KUKA KRL program: MyProgram_209().src

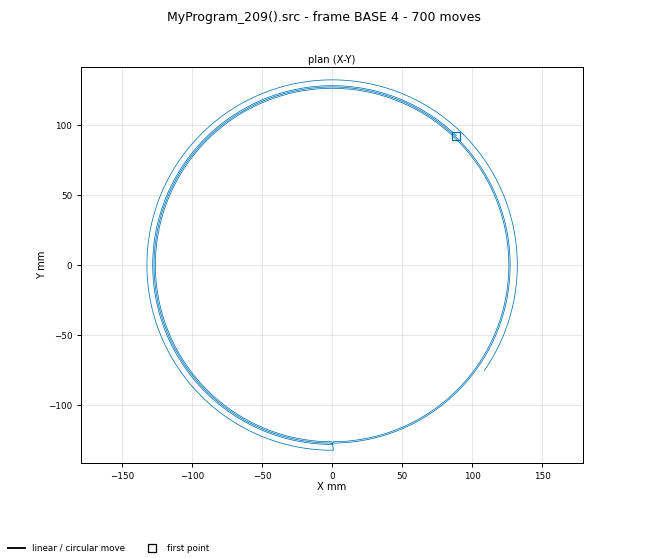
[picture p0: tool path of MyProgram_209().src in frame BASE 4, 700 of 700 moves have a stored position in this frame; points joined in program order, loops and branches not executed]
&ACCESS RVP
&REL 1
&PARAM TEMPLATE = C:\KRC\Roboter\Template\vorgabe
&PARAM EDITMASK = *
DEF MyProgram_209()
; ---- Setting reference (Base) ----
$BASE = BASE_DATA[4]

; --------------------------
; ---- Setting tool (TCP) ----
$TOOL = TOOL_DATA[3]
; --------------------------

$VEL.CP = VEL_APROX_PRINT
Startdeposition()
$VEL.CP = VEL_PRINT
LIN {X 88.7126,Y 92.477,Z 148,A 43.8343,B 21.8486,C -1.1424,E1 21.9863,E2 403.3687} C_DIS
LIN {X 86.374,Y 94.6653,Z 148,A 45.08,B 21.8488,C -1.1368,E1 21.9838,E2 402.1439} C_DIS
LIN {X 83.0937,Y 97.5567,Z 148,A 47.0034,B 21.8488,C -1.1392,E1 21.9797,E2 400.2228} C_DIS
LIN {X 79.622,Y 100.4104,Z 148,A 48.9944,B 21.8486,C -1.1421,E1 21.9754,E2 398.2327} C_DIS
LIN {X 76.1775,Y 103.0485,Z 148,A 50.9778,B 21.8483,C -1.1475,E1 21.971,E2 396.243} C_DIS
LIN {X 72.5158,Y 105.6566,Z 148,A 52.8915,B 21.8483,C -1.1466,E1 21.9666,E2 394.3396} C_DIS
LIN {X 68.9845,Y 107.9954,Z 148,A 54.8188,B 21.8481,C -1.1511,E1 21.9621,E2 392.4074} C_DIS
LIN {X 64.9135,Y 110.4902,Z 148,A 56.7473,B 21.8484,C -1.1451,E1 21.9575,E2 390.5022} C_DIS
LIN {X 61.7494,Y 112.2898,Z 148,A 58.5868,B 21.8478,C -1.1569,E1 21.953,E2 388.6373} C_DIS
LIN {X 58.4226,Y 114.0537,Z 148,A 60.0443,B 21.8482,C -1.149,E1 21.9494,E2 387.2056} C_DIS
LIN {X 55.5123,Y 115.4982,Z 148,A 61.5938,B 21.8479,C -1.1551,E1 21.9455,E2 385.6445} C_DIS
LIN {X 52.3493,Y 116.9655,Z 148,A 63.1517,B 21.8479,C -1.1569,E1 21.9416,E2 384.0863} C_DIS
LIN {X 47.2118,Y 119.1343,Z 148,A 65.6144,B 21.8478,C -1.1582,E1 21.9352,E2 381.627} C_DIS
LIN {X 43.1467,Y 120.6643,Z 148,A 67.6588,B 21.8474,C -1.1646,E1 21.9298,E2 379.5704} C_DIS
LIN {X 39.1405,Y 122.0223,Z 148,A 69.483,B 21.8475,C -1.1632,E1 21.925,E2 377.7539} C_DIS
LIN {X 35.9508,Y 122.9998,Z 148,A 70.9408,B 21.8475,C -1.1628,E1 21.9211,E2 376.3001} C_DIS
LIN {X 32.7097,Y 123.9016,Z 148,A 72.5384,B 21.8473,C -1.168,E1 21.9168,E2 374.6917} C_DIS
LIN {X 28.571,Y 124.9205,Z 148,A 74.3,B 21.8475,C -1.1627,E1 21.9121,E2 372.947} C_DIS
LIN {X 25.5331,Y 125.5767,Z 148,A 75.7516,B 21.8474,C -1.1661,E1 21.9081,E2 371.4884} C_DIS
LIN {X 21.7512,Y 126.2885,Z 148,A 77.403,B 21.8474,C -1.1638,E1 21.9036,E2 369.8455} C_DIS
LIN {X 17.695,Y 126.9194,Z 148,A 79.2772,B 21.8474,C -1.1661,E1 21.8984,E2 367.9672} C_DIS
LIN {X 12.2711,Y 127.5574,Z 148,A 81.7514,B 21.8473,C -1.1679,E1 21.8915,E2 365.49} C_DIS
LIN {X 8.4289,Y 127.87,Z 148,A 83.6291,B 21.8469,C -1.1747,E1 21.8862,E2 363.5952} C_DIS
LIN {X 3.9153,Y 128.0871,Z 148,A 86.0268,B 21.8461,C -1.191,E1 21.8794,E2 361.1544} C_DIS
LIN {X -0.4369,Y 128.146,Z 148,A 87.4571,B 21.8473,C -1.1683,E1 21.8756,E2 359.785} C_DIS
LIN {X -3.2199,Y 128.1064,Z 148,A 89.2919,B 21.846,C -1.1935,E1 21.8703,E2 357.8824} C_DIS
LIN {X -7.9141,Y 127.9018,Z 148,A 90.7155,B 21.8475,C -1.1636,E1 21.8665,E2 356.5386} C_DIS
LIN {X -13.7506,Y 127.4064,Z 148,A 93.443,B 21.8473,C -1.167,E1 21.8589,E2 353.8004} C_DIS
LIN {X -17.7931,Y 126.9054,Z 148,A 95.2356,B 21.8474,C -1.1647,E1 21.854,E2 352.0124} C_DIS
LIN {X -21.7145,Y 126.2946,Z 148,A 97.2457,B 21.847,C -1.1735,E1 21.8483,E2 349.9764} C_DIS
LIN {X -26.441,Y 125.3901,Z 148,A 99.2681,B 21.8474,C -1.1663,E1 21.8429,E2 347.9708} C_DIS
LIN {X -30.0308,Y 124.5776,Z 148,A 100.8142,B 21.8476,C -1.1607,E1 21.8387,E2 346.4374} C_DIS
LIN {X -33.5956,Y 123.6653,Z 148,A 102.571,B 21.8475,C -1.1638,E1 21.8339,E2 344.6693} C_DIS
LIN {X -37.953,Y 122.3977,Z 148,A 105.1421,B 21.8464,C -1.1845,E1 21.8269,E2 342.0373} C_DIS
LIN {X -42.6562,Y 120.8402,Z 148,A 106.8737,B 21.8476,C -1.1614,E1 21.8225,E2 340.364} C_DIS
LIN {X -46.3756,Y 119.46,Z 148,A 108.4825,B 21.8481,C -1.1522,E1 21.8183,E2 338.776} C_DIS
LIN {X -49.6081,Y 118.1544,Z 148,A 110.1026,B 21.8481,C -1.1526,E1 21.8141,E2 337.1506} C_DIS
LIN {X -52.9938,Y 116.6772,Z 148,A 111.8643,B 21.8479,C -1.1548,E1 21.8096,E2 335.3781} C_DIS
LIN {X -56.5469,Y 114.9949,Z 148,A 113.4646,B 21.8484,C -1.1456,E1 21.8056,E2 333.7978} C_DIS
LIN {X -58.9703,Y 113.7731,Z 148,A 114.9346,B 21.848,C -1.1543,E1 21.8019,E2 332.2999} C_DIS
LIN {X -65.619,Y 110.0727,Z 148,A 117.9071,B 21.8491,C -1.1306,E1 21.7949,E2 329.381} C_DIS
LIN {X -68.3515,Y 108.3971,Z 148,A 119.6031,B 21.8487,C -1.1388,E1 21.7907,E2 327.6567} C_DIS
LIN {X -71.7262,Y 106.1943,Z 148,A 121.3334,B 21.8491,C -1.1324,E1 21.7867,E2 325.937} C_DIS
LIN {X -74.857,Y 104.0117,Z 148,A 123.0427,B 21.8492,C -1.1292,E1 21.7828,E2 324.2296} C_DIS
LIN {X -78.0018,Y 101.6738,Z 148,A 125.0863,B 21.8488,C -1.1375,E1 21.7782,E2 322.1549} C_DIS
LIN {X -82.0467,Y 98.4396,Z 148,A 127.2208,B 21.8494,C -1.1251,E1 21.7737,E2 320.0446} C_DIS
LIN {X -84.4392,Y 96.3947,Z 148,A 128.6876,B 21.8494,C -1.1245,E1 21.7706,E2 318.5729} C_DIS
LIN {X -86.7423,Y 94.3273,Z 148,A 130.143,B 21.8494,C -1.1242,E1 21.7675,E2 317.1113} C_DIS
LIN {X -90.1509,Y 91.0754,Z 148,A 132.2112,B 21.8498,C -1.1177,E1 21.7634,E2 315.0505} C_DIS
LIN {X -93.4013,Y 87.739,Z 148,A 134.2865,B 21.85,C -1.1124,E1 21.7594,E2 312.9793} C_DIS
LIN {X -96.9151,Y 83.8411,Z 148,A 136.6811,B 21.8502,C -1.1085,E1 21.755,E2 310.5828} C_DIS
LIN {X -99.8508,Y 80.3225,Z 148,A 139.056,B 21.8498,C -1.1165,E1 21.7507,E2 308.1735} C_DIS
LIN {X -102.2342,Y 77.266,Z 148,A 140.2541,B 21.8511,C -1.0902,E1 21.7488,E2 307.0397} C_DIS
LIN {X -105.1847,Y 73.1985,Z 148,A 142.6997,B 21.8511,C -1.0921,E1 21.7448,E2 304.5749} C_DIS
LIN {X -107.6475,Y 69.5268,Z 148,A 144.6782,B 21.8513,C -1.0867,E1 21.7418,E2 302.5995} C_DIS
LIN {X -111.8681,Y 62.51,Z 148,A 148.3886,B 21.8517,C -1.0783,E1 21.7365,E2 298.8896} C_DIS
LIN {X -113.501,Y 59.4885,Z 148,A 150.8638,B 21.8501,C -1.112,E1 21.7332,E2 296.3079} C_DIS
LIN {X -116.4877,Y 53.4055,Z 148,A 153.0192,B 21.8522,C -1.0675,E1 21.7308,E2 294.2592} C_DIS
LIN {X -118.1611,Y 49.5922,Z 148,A 154.7522,B 21.8527,C -1.0567,E1 21.7289,E2 292.5442} C_DIS
LIN {X -119.4347,Y 46.4407,Z 148,A 157.2556,B 21.851,C -1.0919,E1 21.7263,E2 289.9294} C_DIS
LIN {X -121.6112,Y 40.3995,Z 148,A 160.267,B 21.8512,C -1.0887,E1 21.7236,E2 286.9066} C_DIS
LIN {X -123.6546,Y 33.6359,Z 148,A 162.4583,B 21.8534,C -1.0396,E1 21.722,E2 284.8333} C_DIS
LIN {X -124.5826,Y 30.01,Z 148,A 164.021,B 21.8539,C -1.03,E1 21.721,E2 283.286} C_DIS
LIN {X -125.2863,Y 26.9219,Z 148,A 165.5058,B 21.8539,C -1.0283,E1 21.7201,E2 281.7957} C_DIS
LIN {X -126.0639,Y 23.0116,Z 148,A 167.3491,B 21.8541,C -1.025,E1 21.7191,E2 279.9485} C_DIS
LIN {X -126.7094,Y 19.1419,Z 148,A 169.1664,B 21.8542,C -1.022,E1 21.7183,E2 278.1269} C_DIS
LIN {X -127.217,Y 15.4067,Z 148,A 170.7737,B 21.8546,C -1.0135,E1 21.7178,E2 276.5314} C_DIS
LIN {X -127.626,Y 11.5569,Z 148,A 172.6352,B 21.8546,C -1.0132,E1 21.7173,E2 274.6577} C_DIS
LIN {X -127.9165,Y 7.6748,Z 148,A 174.3037,B 21.855,C -1.0047,E1 21.717,E2 273.0003} C_DIS
LIN {X -128.0928,Y 3.7093,Z 148,A 176.0592,B 21.8553,C -0.9983,E1 21.7168,E2 271.2501} C_DIS
LIN {X -128.1496,Y -0.0528,Z 148,A 178.0622,B 21.8549,C -1.0058,E1 21.7168,E2 269.2128} C_DIS
LIN {X -128.0484,Y -5.0106,Z 148,A -179.9662,B 21.8557,C -0.9889,E1 21.7169,E2 267.2731} C_DIS
LIN {X -127.8019,Y -9.389,Z 148,A -178.0277,B 21.856,C -0.9818,E1 21.7173,E2 265.3402} C_DIS
LIN {X -127.4676,Y -13.1819,Z 148,A -176.2505,B 21.856,C -0.9794,E1 21.7177,E2 263.5571} C_DIS
LIN {X -127.0317,Y -16.8659,Z 148,A -174.6426,B 21.8564,C -0.9721,E1 21.7183,E2 261.9576} C_DIS
LIN {X -126.4164,Y -20.9847,Z 148,A -172.7768,B 21.8566,C -0.9665,E1 21.7191,E2 260.0942} C_DIS
LIN {X -125.7225,Y -24.8164,Z 148,A -170.9204,B 21.8566,C -0.9657,E1 21.7201,E2 258.2272} C_DIS
LIN {X -124.9393,Y -28.4888,Z 148,A -169.3254,B 21.857,C -0.9572,E1 21.721,E2 256.6442} C_DIS
LIN {X -124.0092,Y -32.3059,Z 148,A -167.6182,B 21.8573,C -0.9498,E1 21.7222,E2 254.9454} C_DIS
LIN {X -123.3197,Y -34.8394,Z 148,A -166.2083,B 21.8571,C -0.9558,E1 21.7233,E2 253.5098} C_DIS
LIN {X -122.1023,Y -38.8901,Z 148,A -164.4411,B 21.8575,C -0.9451,E1 21.7247,E2 251.7596} C_DIS
LIN {X -120.0335,Y -44.8704,Z 148,A -161.7574,B 21.8581,C -0.9309,E1 21.7272,E2 249.0967} C_DIS
LIN {X -118.8089,Y -48.0192,Z 148,A -160.1373,B 21.8581,C -0.9309,E1 21.7289,E2 247.4659} C_DIS
LIN {X -117.5359,Y -51.0561,Z 148,A -158.593,B 21.8581,C -0.9297,E1 21.7306,E2 245.9152} C_DIS
LIN {X -115.7831,Y -54.9159,Z 148,A -156.6975,B 21.8584,C -0.9243,E1 21.7328,E2 244.0221} C_DIS
LIN {X -114.2963,Y -57.9462,Z 148,A -155.3639,B 21.8588,C -0.913,E1 21.7344,E2 242.7107} C_DIS
LIN {X -112.3675,Y -61.6074,Z 148,A -153.2902,B 21.8587,C -0.917,E1 21.7372,E2 240.6134} C_DIS
LIN {X -110.1286,Y -65.5253,Z 148,A -151.2391,B 21.8588,C -0.913,E1 21.7401,E2 238.5607} C_DIS
LIN {X -107.9003,Y -69.1332,Z 148,A -149.3445,B 21.859,C -0.908,E1 21.7429,E2 236.6684} C_DIS
LIN {X -105.4709,Y -72.7864,Z 148,A -147.3415,B 21.8591,C -0.9048,E1 21.746,E2 234.6627} C_DIS
LIN {X -103.0791,Y -76.1358,Z 148,A -145.2043,B 21.8588,C -0.9125,E1 21.7496,E2 232.4926} C_DIS
LIN {X -100.9621,Y -78.9203,Z 148,A -143.8505,B 21.8593,C -0.9001,E1 21.7519,E2 231.165} C_DIS
LIN {X -97.9265,Y -82.6583,Z 148,A -141.7279,B 21.8596,C -0.8938,E1 21.7557,E2 229.0479} C_DIS
LIN {X -94.8508,Y -86.1696,Z 148,A -139.6882,B 21.8598,C -0.8871,E1 21.7594,E2 227.0156} C_DIS
LIN {X -91.854,Y -89.3577,Z 148,A -137.6716,B 21.8599,C -0.8854,E1 21.7633,E2 224.9936} C_DIS
LIN {X -88.8005,Y -92.3929,Z 148,A -135.7075,B 21.8599,C -0.883,E1 21.7673,E2 223.0264} C_DIS
LIN {X -85.5251,Y -95.4322,Z 148,A -133.7701,B 21.8602,C -0.8765,E1 21.7712,E2 221.0975} C_DIS
LIN {X -82.2328,Y -98.2836,Z 148,A -131.8219,B 21.8604,C -0.8728,E1 21.7754,E2 219.1505} C_DIS
LIN {X -78.9585,Y -100.9331,Z 148,A -129.8981,B 21.8604,C -0.871,E1 21.7796,E2 217.2231} C_DIS
LIN {X -76.531,Y -102.7855,Z 148,A -128.228,B 21.8601,C -0.8814,E1 21.7834,E2 215.5179} C_DIS
LIN {X -73.5721,Y -104.9244,Z 148,A -126.8123,B 21.8605,C -0.8696,E1 21.7866,E2 214.1286} C_DIS
LIN {X -69.6016,Y -107.5989,Z 148,A -124.607,B 21.8605,C -0.8689,E1 21.7917,E2 211.9167} C_DIS
LIN {X -66.4857,Y -109.5516,Z 148,A -122.9155,B 21.8605,C -0.8684,E1 21.7958,E2 210.2204} C_DIS
LIN {X -61.9331,Y -112.1881,Z 148,A -120.7457,B 21.861,C -0.8574,E1 21.801,E2 208.0729} C_DIS
LIN {X -58.4074,Y -114.0615,Z 148,A -119.0154,B 21.8611,C -0.8528,E1 21.8053,E2 206.3495} C_DIS
LIN {X -55.4723,Y -115.5174,Z 148,A -117.5903,B 21.8613,C -0.8493,E1 21.8088,E2 204.9296} C_DIS
LIN {X -52.5672,Y -116.868,Z 148,A -115.934,B 21.861,C -0.8573,E1 21.8131,E2 203.2472} C_DIS
LIN {X -48.8863,Y -118.4559,Z 148,A -114.0372,B 21.8609,C -0.8598,E1 21.818,E2 201.3383} C_DIS
LIN {X -43.8696,Y -120.4036,Z 148,A -111.8803,B 21.8614,C -0.8469,E1 21.8236,E2 199.2112} C_DIS
LIN {X -40.6809,Y -121.5175,Z 148,A -110.4068,B 21.8614,C -0.844,E1 21.8275,E2 197.742} C_DIS
LIN {X -37.5286,Y -122.5276,Z 148,A -108.9305,B 21.8615,C -0.8428,E1 21.8314,E2 196.2662} C_DIS
LIN {X -34.3559,Y -123.4549,Z 148,A -107.4414,B 21.8615,C -0.8422,E1 21.8354,E2 194.7757} C_DIS
LIN {X -30.9895,Y -124.3438,Z 148,A -105.749,B 21.8613,C -0.8472,E1 21.84,E2 193.0672} C_DIS
LIN {X -27.2663,Y -125.212,Z 148,A -104.1471,B 21.8615,C -0.8417,E1 21.8444,E2 191.4777} C_DIS
LIN {X -23.6613,Y -125.9434,Z 148,A -102.2747,B 21.8612,C -0.8509,E1 21.8496,E2 189.578} C_DIS
LIN {X -19.0769,Y -126.7194,Z 148,A -99.8973,B 21.8607,C -0.8634,E1 21.8562,E2 187.1647} C_DIS
LIN {X -14.7427,Y -127.2962,Z 148,A -98.4357,B 21.8616,C -0.8414,E1 21.8601,E2 185.7612} C_DIS
LIN {X -8.5481,Y -127.8627,Z 148,A -95.7698,B 21.8617,C -0.8361,E1 21.8675,E2 183.1081} C_DIS
LIN {X -2.0512,Y -128.13,Z 148,A -92.7229,B 21.8615,C -0.8425,E1 21.8761,E2 180.0434} C_DIS
LIN {X 0.9079,Y -128.1328,Z 148,A -91.2252,B 21.8612,C -0.8507,E1 21.8803,E2 178.5239} C_DIS
Enddeposition()
LIN {X 0.9079,Y -128.1328,Z 148,A -91.2252,B 21.8612,C -0.8507,E1 21.8803,E2 178.5239} C_DIS
Startdeposition()
$VEL.CP = VEL_PRINT
LIN {X -0.6648,Y -127.1927,Z 148,A -92.5574,B 20.775,C -0.658,E1 20.7835,E2 180.2621} C_DIS
LIN {X -5.688,Y -127.069,Z 148,A -94.7279,B 20.775,C -0.6615,E1 20.7774,E2 182.4229} C_DIS
LIN {X -10.6847,Y -126.7448,Z 148,A -97.0594,B 20.775,C -0.6585,E1 20.7709,E2 184.764} C_DIS
LIN {X -13.7804,Y -126.4457,Z 148,A -98.4019,B 20.775,C -0.661,E1 20.7672,E2 186.1003} C_DIS
LIN {X -17.6557,Y -125.9634,Z 148,A -100.0322,B 20.7748,C -0.6666,E1 20.7627,E2 187.7162} C_DIS
LIN {X -20.443,Y -125.5416,Z 148,A -101.5759,B 20.7751,C -0.6559,E1 20.7584,E2 189.2918} C_DIS
LIN {X -24.2382,Y -124.8639,Z 148,A -103.3206,B 20.7751,C -0.6563,E1 20.7536,E2 191.0377} C_DIS
LIN {X -28.3968,Y -123.9838,Z 148,A -105.0923,B 20.7749,C -0.6629,E1 20.7488,E2 192.7933} C_DIS
LIN {X -31.4491,Y -123.245,Z 148,A -106.5561,B 20.7749,C -0.6618,E1 20.7448,E2 194.2629} C_DIS
LIN {X -34.5303,Y -122.4176,Z 148,A -107.9467,B 20.7749,C -0.6646,E1 20.7411,E2 195.6483} C_DIS
LIN {X -38.0472,Y -121.3722,Z 148,A -109.7467,B 20.7749,C -0.6599,E1 20.7362,E2 197.4653} C_DIS
LIN {X -41.7936,Y -120.1317,Z 148,A -111.4421,B 20.7749,C -0.6647,E1 20.7318,E2 199.1511} C_DIS
LIN {X -44.7587,Y -119.0588,Z 148,A -112.8824,B 20.7749,C -0.6652,E1 20.728,E2 200.5935} C_DIS
LIN {X -47.7996,Y -117.871,Z 148,A -114.3557,B 20.7748,C -0.6665,E1 20.7242,E2 202.067} C_DIS
LIN {X -51.6255,Y -116.2463,Z 148,A -116.2801,B 20.7748,C -0.6665,E1 20.7192,E2 203.9972} C_DIS
LIN {X -55.133,Y -114.6244,Z 148,A -117.975,B 20.7747,C -0.6703,E1 20.715,E2 205.6864} C_DIS
LIN {X -58.7811,Y -112.7972,Z 148,A -119.8364,B 20.7747,C -0.6717,E1 20.7103,E2 207.55} C_DIS
LIN {X -62.6527,Y -110.6958,Z 148,A -121.9529,B 20.7747,C -0.6692,E1 20.7051,E2 209.6811} C_DIS
LIN {X -66.3485,Y -108.5204,Z 148,A -123.7887,B 20.7745,C -0.6758,E1 20.7007,E2 211.5052} C_DIS
LIN {X -69.1373,Y -106.7653,Z 148,A -125.3261,B 20.7745,C -0.676,E1 20.6971,E2 213.048} C_DIS
LIN {X -75.751,Y -102.1784,Z 148,A -128.8248,B 20.7741,C -0.6869,E1 20.6892,E2 216.5305} C_DIS
LIN {X -78.7864,Y -99.8577,Z 148,A -130.6927,B 20.7742,C -0.6843,E1 20.685,E2 218.4142} C_DIS
LIN {X -82.1364,Y -97.121,Z 148,A -132.6306,B 20.7741,C -0.6883,E1 20.6808,E2 220.3497} C_DIS
LIN {X -85.2092,Y -94.4366,Z 148,A -134.5328,B 20.7741,C -0.6895,E1 20.6769,E2 222.2581} C_DIS
LIN {X -88.5102,Y -91.3494,Z 148,A -136.5341,B 20.7739,C -0.695,E1 20.6728,E2 224.2539} C_DIS
LIN {X -91.5331,Y -88.3205,Z 148,A -138.4406,B 20.7737,C -0.6998,E1 20.6691,E2 226.1566} C_DIS
LIN {X -94.4543,Y -85.1898,Z 148,A -140.4411,B 20.7737,C -0.7013,E1 20.6653,E2 228.1637} C_DIS
LIN {X -97.3497,Y -81.8647,Z 148,A -142.4032,B 20.7735,C -0.7068,E1 20.6618,E2 230.1213} C_DIS
LIN {X -102.4162,Y -75.4302,Z 148,A -145.9407,B 20.773,C -0.7213,E1 20.6557,E2 233.6383} C_DIS
LIN {X -104.2844,Y -72.8258,Z 148,A -147.5893,B 20.7732,C -0.7171,E1 20.653,E2 235.3087} C_DIS
LIN {X -106.7797,Y -69.1151,Z 148,A -149.5998,B 20.773,C -0.7223,E1 20.6499,E2 237.3167} C_DIS
LIN {X -108.9775,Y -65.5954,Z 148,A -151.4874,B 20.7729,C -0.7265,E1 20.6472,E2 239.2045} C_DIS
LIN {X -111.0679,Y -61.9906,Z 148,A -153.3612,B 20.7727,C -0.7316,E1 20.6446,E2 241.0758} C_DIS
LIN {X -113.0767,Y -58.2435,Z 148,A -155.114,B 20.7723,C -0.7429,E1 20.6423,E2 242.808} C_DIS
LIN {X -114.6357,Y -55.1093,Z 148,A -156.8307,B 20.7723,C -0.742,E1 20.6402,E2 244.5386} C_DIS
LIN {X -116.2149,Y -51.6958,Z 148,A -158.5043,B 20.7721,C -0.7475,E1 20.6383,E2 246.2079} C_DIS
LIN {X -117.8026,Y -47.9692,Z 148,A -160.4669,B 20.7721,C -0.7475,E1 20.6362,E2 248.1838} C_DIS
LIN {X -119.2228,Y -44.3209,Z 148,A -163.0045,B 20.7729,C -0.724,E1 20.6336,E2 250.8057} C_DIS
LIN {X -121.1824,Y -38.6412,Z 148,A -164.4761,B 20.7711,C -0.7777,E1 20.6325,E2 252.1352} C_DIS
LIN {X -122.7146,Y -33.4661,Z 148,A -167.2451,B 20.7713,C -0.7723,E1 20.6303,E2 254.9394} C_DIS
LIN {X -123.5827,Y -30.0959,Z 148,A -168.9047,B 20.7713,C -0.7736,E1 20.6291,E2 256.6071} C_DIS
LIN {X -124.346,Y -26.7661,Z 148,A -170.4313,B 20.771,C -0.7787,E1 20.6282,E2 258.1302} C_DIS
LIN {X -125.1283,Y -22.8357,Z 148,A -172.324,B 20.771,C -0.781,E1 20.6272,E2 260.0302} C_DIS
LIN {X -125.7464,Y -19.1394,Z 148,A -174.0513,B 20.7708,C -0.7848,E1 20.6264,E2 261.7594} C_DIS
LIN {X -126.2921,Y -15.1223,Z 148,A -175.793,B 20.7705,C -0.7936,E1 20.6258,E2 263.4889} C_DIS
LIN {X -126.6752,Y -11.4994,Z 148,A -177.5058,B 20.7705,C -0.796,E1 20.6253,E2 265.2074} C_DIS
LIN {X -126.9566,Y -7.7738,Z 148,A -179.1506,B 20.7702,C -0.8028,E1 20.625,E2 266.8453} C_DIS
LIN {X -127.1313,Y -4.0387,Z 148,A 179.0349,B 20.7702,C -0.8032,E1 20.6248,E2 268.6718} C_DIS
LIN {X -127.1976,Y -0.0192,Z 148,A 177.1579,B 20.77,C -0.8065,E1 20.6248,E2 270.5536} C_DIS
LIN {X -127.1309,Y 4.0542,Z 148,A 175.4305,B 20.7697,C -0.8163,E1 20.6249,E2 272.2659} C_DIS
LIN {X -126.9529,Y 7.8336,Z 148,A 173.7492,B 20.7694,C -0.8225,E1 20.6252,E2 273.9419} C_DIS
LIN {X -126.6591,Y 11.6669,Z 148,A 171.9608,B 20.7694,C -0.8259,E1 20.6256,E2 275.734} C_DIS
LIN {X -126.2598,Y 15.3937,Z 148,A 170.315,B 20.769,C -0.8328,E1 20.6261,E2 277.3723} C_DIS
LIN {X -125.7312,Y 19.2379,Z 148,A 168.5125,B 20.769,C -0.8363,E1 20.6268,E2 279.1781} C_DIS
LIN {X -125.1256,Y 22.8507,Z 148,A 166.7747,B 20.7688,C -0.8382,E1 20.6277,E2 280.9231} C_DIS
LIN {X -124.3198,Y 26.8875,Z 148,A 164.9973,B 20.7685,C -0.8469,E1 20.6287,E2 282.6888} C_DIS
LIN {X -123.3924,Y 30.8683,Z 148,A 162.652,B 20.769,C -0.8341,E1 20.6303,E2 285.0873} C_DIS
LIN {X -122.2778,Y 35.0289,Z 148,A 161.1134,B 20.7682,C -0.8548,E1 20.6314,E2 286.5782} C_DIS
LIN {X -121.2023,Y 38.579,Z 148,A 159.4896,B 20.7679,C -0.8616,E1 20.6327,E2 288.1939} C_DIS
LIN {X -119.9994,Y 42.1752,Z 148,A 157.4991,B 20.7681,C -0.8564,E1 20.6346,E2 290.2131} C_DIS
LIN {X -118.8852,Y 45.222,Z 148,A 156.3939,B 20.7674,C -0.8739,E1 20.6356,E2 291.2763} C_DIS
LIN {X -117.8921,Y 47.7473,Z 148,A 155.1011,B 20.7674,C -0.875,E1 20.637,E2 292.575} C_DIS
LIN {X -116.6356,Y 50.7397,Z 148,A 153.603,B 20.7673,C -0.878,E1 20.6386,E2 294.0747} C_DIS
LIN {X -114.2482,Y 55.9087,Z 148,A 151.2271,B 20.7667,C -0.8925,E1 20.6414,E2 296.4254} C_DIS
LIN {X -112.4662,Y 59.4116,Z 148,A 149.3018,B 20.7667,C -0.8919,E1 20.6439,E2 298.3652} C_DIS
LIN {X -110.6699,Y 62.6985,Z 148,A 147.4266,B 20.7667,C -0.8896,E1 20.6464,E2 300.2588} C_DIS
LIN {X -107.6888,Y 67.6901,Z 148,A 145.092,B 20.766,C -0.9075,E1 20.6498,E2 302.5574} C_DIS
LIN {X -106.0207,Y 70.2747,Z 148,A 143.4229,B 20.7663,C -0.9007,E1 20.6524,E2 304.2562} C_DIS
LIN {X -103.2772,Y 74.2476,Z 148,A 141.3113,B 20.766,C -0.9089,E1 20.6557,E2 306.3573} C_DIS
LIN {X -101.0954,Y 77.1913,Z 148,A 139.5502,B 20.766,C -0.9091,E1 20.6587,E2 308.1282} C_DIS
LIN {X -98.8233,Y 80.08,Z 148,A 137.9226,B 20.7658,C -0.9144,E1 20.6615,E2 309.7502} C_DIS
LIN {X -94.0564,Y 85.6283,Z 148,A 134.8835,B 20.765,C -0.9321,E1 20.667,E2 312.7558} C_DIS
LIN {X -91.8901,Y 87.9488,Z 148,A 133.1801,B 20.7653,C -0.9253,E1 20.6703,E2 314.4877} C_DIS
LIN {X -89.0135,Y 90.859,Z 148,A 130.8639,B 20.7659,C -0.9119,E1 20.6751,E2 316.8539} C_DIS
LIN {X -85.8449,Y 93.859,Z 148,A 129.3119,B 20.765,C -0.9318,E1 20.6781,E2 318.3571} C_DIS
LIN {X -82.652,Y 96.6827,Z 148,A 127.3834,B 20.7648,C -0.9357,E1 20.6822,E2 320.2839} C_DIS
LIN {X -79.4153,Y 99.3582,Z 148,A 124.9268,B 20.7656,C -0.9184,E1 20.6877,E2 322.8006} C_DIS
LIN {X -75.4783,Y 102.3808,Z 148,A 123.3533,B 20.7643,C -0.9479,E1 20.691,E2 324.2976} C_DIS
LIN {X -71.4179,Y 105.2534,Z 148,A 120.9885,B 20.7643,C -0.9475,E1 20.6965,E2 326.6735} C_DIS
LIN {X -67.6901,Y 107.6888,Z 148,A 118.9964,B 20.7642,C -0.9517,E1 20.7011,E2 328.6616} C_DIS
LIN {X -59.0803,Y 112.6401,Z 148,A 114.6834,B 20.7635,C -0.9654,E1 20.7116,E2 332.9512} C_DIS
LIN {X -56.4309,Y 113.9906,Z 148,A 113.1516,B 20.7638,C -0.9601,E1 20.7154,E2 334.503} C_DIS
LIN {X -52.7447,Y 115.7444,Z 148,A 111.3758,B 20.7636,C -0.9652,E1 20.7199,E2 336.2699} C_DIS
LIN {X -49.4758,Y 117.178,Z 148,A 109.74,B 20.7636,C -0.9664,E1 20.7241,E2 337.9071} C_DIS
LIN {X -46.105,Y 118.5438,Z 148,A 108.1164,B 20.7634,C -0.9691,E1 20.7283,E2 339.5273} C_DIS
LIN {X -42.7288,Y 119.803,Z 148,A 106.3737,B 20.7635,C -0.9665,E1 20.7329,E2 341.2818} C_DIS
LIN {X -37.6788,Y 121.486,Z 148,A 104.2543,B 20.7629,C -0.98,E1 20.7384,E2 343.3678} C_DIS
LIN {X -33.9288,Y 122.5858,Z 148,A 102.2739,B 20.7632,C -0.9732,E1 20.7438,E2 345.3712} C_DIS
LIN {X -30.0369,Y 123.5969,Z 148,A 100.4757,B 20.7632,C -0.9754,E1 20.7487,E2 347.1665} C_DIS
LIN {X -26.4495,Y 124.4144,Z 148,A 98.8829,B 20.7629,C -0.9793,E1 20.753,E2 348.7506} C_DIS
LIN {X -21.3035,Y 125.398,Z 148,A 96.4295,B 20.763,C -0.9773,E1 20.7598,E2 351.2127} C_DIS
LIN {X -17.2898,Y 126.0157,Z 148,A 94.5257,B 20.763,C -0.9755,E1 20.765,E2 353.1236} C_DIS
LIN {X -13.2816,Y 126.4994,Z 148,A 92.584,B 20.7633,C -0.9715,E1 20.7705,E2 355.0779} C_DIS
LIN {X -8.2031,Y 126.9302,Z 148,A 90.331,B 20.7632,C -0.9741,E1 20.7767,E2 357.3247} C_DIS
LIN {X -3.3992,Y 127.1491,Z 148,A 88.414,B 20.7627,C -0.9846,E1 20.782,E2 359.2125} C_DIS
LIN {X -0.2495,Y 127.195,Z 148,A 86.7618,B 20.7631,C -0.9756,E1 20.7867,E2 360.8902} C_DIS
LIN {X 4.5654,Y 127.1131,Z 148,A 84.733,B 20.7628,C -0.9813,E1 20.7923,E2 362.9022} C_DIS
LIN {X 8.479,Y 126.9132,Z 148,A 82.8948,B 20.763,C -0.9783,E1 20.7974,E2 364.7481} C_DIS
LIN {X 12.6954,Y 126.5603,Z 148,A 80.8686,B 20.7632,C -0.9732,E1 20.8031,E2 366.787} C_DIS
LIN {X 17.3436,Y 126.008,Z 148,A 78.9712,B 20.7628,C -0.9812,E1 20.8083,E2 368.6601} C_DIS
LIN {X 20.9767,Y 125.4526,Z 148,A 77.3366,B 20.7628,C -0.9815,E1 20.8128,E2 370.2918} C_DIS
LIN {X 24.7369,Y 124.7672,Z 148,A 75.5499,B 20.763,C -0.9781,E1 20.8177,E2 372.0856} C_DIS
LIN {X 28.4264,Y 123.977,Z 148,A 73.982,B 20.7628,C -0.9826,E1 20.822,E2 373.6383} C_DIS
LIN {X 31.5493,Y 123.2195,Z 148,A 72.5628,B 20.7628,C -0.9829,E1 20.8258,E2 375.0542} C_DIS
LIN {X 34.8468,Y 122.3291,Z 148,A 70.8482,B 20.7631,C -0.9746,E1 20.8305,E2 376.7886} C_DIS
LIN {X 38.7331,Y 121.1531,Z 148,A 69.1305,B 20.763,C -0.9777,E1 20.835,E2 378.4937} C_DIS
LIN {X 41.8208,Y 120.1223,Z 148,A 67.6304,B 20.7631,C -0.975,E1 20.839,E2 379.9976} C_DIS
LIN {X 45.0138,Y 118.9632,Z 148,A 66.1442,B 20.7631,C -0.9754,E1 20.8429,E2 381.479} C_DIS
LIN {X 48.8551,Y 117.4372,Z 148,A 64.2783,B 20.7631,C -0.9733,E1 20.8477,E2 383.3456} C_DIS
LIN {X 51.9103,Y 116.119,Z 148,A 62.7803,B 20.7633,C -0.9716,E1 20.8515,E2 384.8437} C_DIS
LIN {X 54.7965,Y 114.7851,Z 148,A 61.3247,B 20.7633,C -0.969,E1 20.8552,E2 386.3023} C_DIS
LIN {X 58.4037,Y 112.9951,Z 148,A 59.4176,B 20.7637,C -0.9627,E1 20.86,E2 388.2205} C_DIS
LIN {X 62.6631,Y 110.6899,Z 148,A 57.3932,B 20.7635,C -0.9662,E1 20.8649,E2 390.2277} C_DIS
LIN {X 66.0176,Y 108.7222,Z 148,A 55.5892,B 20.7637,C -0.9615,E1 20.8692,E2 392.0383} C_DIS
LIN {X 69.2713,Y 106.6783,Z 148,A 53.8368,B 20.7639,C -0.9579,E1 20.8734,E2 393.7939} C_DIS
LIN {X 72.9716,Y 104.1829,Z 148,A 51.7789,B 20.7641,C -0.9525,E1 20.8781,E2 395.8582} C_DIS
LIN {X 76.5305,Y 101.5966,Z 148,A 49.8402,B 20.7641,C -0.9509,E1 20.8825,E2 397.793} C_DIS
LIN {X 80.1422,Y 98.7731,Z 148,A 47.7701,B 20.7644,C -0.9469,E1 20.887,E2 399.8649} C_DIS
LIN {X 83.421,Y 96.0197,Z 148,A 45.8398,B 20.7645,C -0.9431,E1 20.8911,E2 401.7966} C_DIS
LIN {X 86.8478,Y 92.9316,Z 148,A 43.9099,B 20.7645,C -0.9452,E1 20.895,E2 403.7109} C_DIS
LIN {X 89.5534,Y 90.3271,Z 148,A 42.1887,B 20.7646,C -0.9404,E1 20.8985,E2 405.4368} C_DIS
LIN {X 92.5082,Y 87.2984,Z 148,A 40.4133,B 20.7646,C -0.9418,E1 20.9019,E2 407.1988} C_DIS
LIN {X 94.8817,Y 84.7128,Z 148,A 38.6755,B 20.765,C -0.9316,E1 20.9052,E2 408.9557} C_DIS
LIN {X 97.6473,Y 81.51,Z 148,A 36.7736,B 20.7652,C -0.9274,E1 20.9086,E2 410.8588} C_DIS
LIN {X 100.2918,Y 78.2335,Z 148,A 34.8442,B 20.7655,C -0.9215,E1 20.912,E2 412.7937} C_DIS
LIN {X 102.7728,Y 74.9443,Z 148,A 32.9867,B 20.7657,C -0.9169,E1 20.9151,E2 414.6531} C_DIS
LIN {X 105.3268,Y 71.3095,Z 148,A 31.1017,B 20.7657,C -0.9169,E1 20.9181,E2 416.5268} C_DIS
LIN {X 107.3544,Y 68.22,Z 148,A 29.4155,B 20.7659,C -0.9116,E1 20.9206,E2 418.2172} C_DIS
LIN {X 109.7097,Y 64.3628,Z 148,A 27.3515,B 20.7661,C -0.9051,E1 20.9236,E2 420.2866} C_DIS
LIN {X 111.8555,Y 60.5581,Z 148,A 25.4113,B 20.7663,C -0.901,E1 20.9262,E2 422.2259} C_DIS
LIN {X 113.4538,Y 57.5028,Z 148,A 23.9559,B 20.7663,C -0.901,E1 20.9281,E2 423.6718} C_DIS
LIN {X 115.0078,Y 54.3305,Z 148,A 22.386,B 20.7665,C -0.8975,E1 20.93,E2 425.2412} C_DIS
LIN {X 116.6075,Y 50.8045,Z 148,A 20.157,B 20.7675,C -0.8716,E1 20.9325,E2 427.5277} C_DIS
LIN {X 118.2232,Y 46.9257,Z 148,A 18.8245,B 20.7668,C -0.8904,E1 20.9339,E2 428.7986} C_DIS
LIN {X 119.4775,Y 43.6316,Z 148,A 17.3192,B 20.7668,C -0.8894,E1 20.9353,E2 430.2963} C_DIS
LIN {X 120.7143,Y 40.0796,Z 148,A 15.5157,B 20.7672,C -0.8797,E1 20.937,E2 432.1146} C_DIS
LIN {X 121.8566,Y 36.4675,Z 148,A 13.7185,B 20.7676,C -0.8706,E1 20.9385,E2 433.9246} C_DIS
LIN {X 122.9188,Y 32.7003,Z 148,A 12.0702,B 20.7676,C -0.8704,E1 20.9397,E2 435.562} C_DIS
LIN {X 123.825,Y 29.0905,Z 148,A 10.2871,B 20.768,C -0.8606,E1 20.9409,E2 437.3599} C_DIS
LIN {X 124.6388,Y 25.3677,Z 148,A 8.687,B 20.768,C -0.8605,E1 20.9418,E2 438.9488} C_DIS
LIN {X 125.3082,Y 21.8301,Z 148,A 7.0724,B 20.7681,C -0.8558,E1 20.9426,E2 440.565} C_DIS
LIN {X 125.9648,Y 17.6454,Z 148,A 5.0685,B 20.7685,C -0.8457,E1 20.9434,E2 442.5827} C_DIS
LIN {X 126.6382,Y 11.8838,Z 148,A 2.6958,B 20.7685,C -0.8481,E1 20.9442,E2 444.9315} C_DIS
LIN {X 126.8677,Y 9.1107,Z 148,A 1.3449,B 20.7688,C -0.8398,E1 20.9444,E2 446.2956} C_DIS
LIN {X 127.1077,Y 4.7035,Z 148,A -0.8917,B 20.7694,C -0.8227,E1 20.9447,E2 448.5639} C_DIS
LIN {X 127.1968,Y 0.1898,Z 148,A -2.7124,B 20.7694,C -0.8256,E1 20.9447,E2 450.3634} C_DIS
LIN {X 127.1471,Y -3.4693,Z 148,A -4.2603,B 20.7694,C -0.8248,E1 20.9447,E2 451.902} C_DIS
LIN {X 126.9264,Y -8.2634,Z 148,A -6.3488,B 20.7694,C -0.8212,E1 20.9444,E2 453.9855} C_DIS
LIN {X 126.7051,Y -11.154,Z 148,A -7.9398,B 20.7701,C -0.8045,E1 20.944,E2 455.6116} C_DIS
LIN {X 126.2648,Y -15.3511,Z 148,A -9.548,B 20.7698,C -0.8113,E1 20.9435,E2 457.1889} C_DIS
LIN {X 125.8842,Y -18.2098,Z 148,A -10.8413,B 20.77,C -0.8075,E1 20.943,E2 458.4837} C_DIS
LIN {X 125.197,Y -22.4517,Z 148,A -12.6111,B 20.77,C -0.8087,E1 20.9422,E2 460.2374} C_DIS
LIN {X 124.6608,Y -25.2597,Z 148,A -14.0854,B 20.7704,C -0.7964,E1 20.9414,E2 461.7354} C_DIS
LIN {X 123.9272,Y -28.6443,Z 148,A -15.674,B 20.7706,C -0.7903,E1 20.9404,E2 463.3299} C_DIS
LIN {X 122.9754,Y -32.4879,Z 148,A -17.4549,B 20.7708,C -0.7849,E1 20.9392,E2 465.1133} C_DIS
LIN {X 121.9527,Y -36.1393,Z 148,A -19.0286,B 20.7708,C -0.7855,E1 20.938,E2 466.6742} C_DIS
LIN {X 121.1677,Y -38.6875,Z 148,A -20.285,B 20.771,C -0.7794,E1 20.9369,E2 467.939} C_DIS
LIN {X 120.0837,Y -41.9319,Z 148,A -21.8685,B 20.7713,C -0.7728,E1 20.9355,E2 469.5299} C_DIS
LIN {X 118.9812,Y -44.9657,Z 148,A -23.2457,B 20.7713,C -0.7718,E1 20.9342,E2 470.9006} C_DIS
LIN {X 117.5175,Y -48.663,Z 148,A -25.053,B 20.7715,C -0.7657,E1 20.9323,E2 472.7127} C_DIS
LIN {X 116.1506,Y -51.8396,Z 148,A -26.5945,B 20.7716,C -0.7618,E1 20.9306,E2 474.2549} C_DIS
LIN {X 114.4587,Y -55.4799,Z 148,A -28.3597,B 20.7718,C -0.7583,E1 20.9285,E2 476.018} C_DIS
LIN {X 112.502,Y -59.3433,Z 148,A -30.1504,B 20.7718,C -0.7597,E1 20.9262,E2 477.7932} C_DIS
LIN {X 110.8729,Y -62.3377,Z 148,A -31.9453,B 20.7723,C -0.7439,E1 20.9237,E2 479.6208} C_DIS
LIN {X 108.6701,Y -66.1037,Z 148,A -33.8906,B 20.7724,C -0.7393,E1 20.9209,E2 481.5669} C_DIS
LIN {X 106.249,Y -69.928,Z 148,A -35.8531,B 20.7724,C -0.737,E1 20.918,E2 483.5238} C_DIS
LIN {X 104.0993,Y -73.0902,Z 148,A -37.5794,B 20.7727,C -0.7321,E1 20.9152,E2 485.2532} C_DIS
LIN {X 101.8393,Y -76.2077,Z 148,A -39.5586,B 20.7732,C -0.7169,E1 20.9119,E2 487.2634} C_DIS
LIN {X 99.8694,Y -78.7714,Z 148,A -40.4832,B 20.7725,C -0.7362,E1 20.9104,E2 488.1286} C_DIS
LIN {X 96.8418,Y -82.4648,Z 148,A -42.9219,B 20.7731,C -0.7182,E1 20.906,E2 490.6039} C_DIS
LIN {X 93.6109,Y -86.1148,Z 148,A -45.3326,B 20.7736,C -0.7035,E1 20.9014,E2 493.0428} C_DIS
LIN {X 91.3613,Y -88.4979,Z 148,A -46.4872,B 20.7733,C -0.7138,E1 20.8993,E2 494.1623} C_DIS
LIN {X 88.638,Y -91.2256,Z 148,A -48.3029,B 20.7735,C -0.7063,E1 20.8956,E2 495.9898} C_DIS
LIN {X 84.6186,Y -94.9658,Z 148,A -50.8332,B 20.7738,C -0.6982,E1 20.8904,E2 498.5302} C_DIS
LIN {X 81.3838,Y -97.7525,Z 148,A -52.661,B 20.7738,C -0.6981,E1 20.8865,E2 500.3496} C_DIS
LIN {X 78.1396,Y -100.3646,Z 148,A -54.5596,B 20.7739,C -0.6931,E1 20.8824,E2 502.2533} C_DIS
LIN {X 74.0707,Y -103.4036,Z 148,A -56.7803,B 20.7739,C -0.6914,E1 20.8774,E2 504.4694} C_DIS
LIN {X 70.7487,Y -105.7044,Z 148,A -58.6078,B 20.7741,C -0.6875,E1 20.8731,E2 506.3} C_DIS
LIN {X 67.4938,Y -107.8123,Z 148,A -61.0755,B 20.7752,C -0.6537,E1 20.8671,E2 508.853} C_DIS
LIN {X 62.6083,Y -110.7208,Z 148,A -62.6137,B 20.774,C -0.6926,E1 20.8637,E2 510.2763} C_DIS
LIN {X 58.9355,Y -112.7162,Z 148,A -64.7226,B 20.7744,C -0.6798,E1 20.8584,E2 512.4136} C_DIS
LIN {X 55.9119,Y -114.2467,Z 148,A -66.3193,B 20.7745,C -0.6744,E1 20.8544,E2 514.0202} C_DIS
LIN {X 50.2698,Y -116.8387,Z 148,A -68.9815,B 20.7745,C -0.676,E1 20.8477,E2 516.6699} C_DIS
LIN {X 47.191,Y -118.1163,Z 148,A -70.455,B 20.7745,C -0.6751,E1 20.8438,E2 518.1417} C_DIS
LIN {X 44.1575,Y -119.2839,Z 148,A -71.9514,B 20.7746,C -0.6718,E1 20.8399,E2 519.6433} C_DIS
LIN {X 39.121,Y -121.0292,Z 148,A -74.258,B 20.7746,C -0.6729,E1 20.8339,E2 521.9413} C_DIS
LIN {X 35.9646,Y -122.0038,Z 148,A -75.8767,B 20.7748,C -0.6658,E1 20.8295,E2 523.5765} C_DIS
LIN {X 32.4348,Y -122.9896,Z 148,A -77.6132,B 20.775,C -0.6605,E1 20.8248,E2 525.3245} C_DIS
LIN {X 28.5115,Y -123.9576,Z 148,A -79.3182,B 20.7749,C -0.6636,E1 20.8202,E2 527.0176} C_DIS
LIN {X 25.0595,Y -124.7015,Z 148,A -80.8798,B 20.7749,C -0.6636,E1 20.8159,E2 528.5772} C_DIS
LIN {X 20.7644,Y -125.488,Z 148,A -83.2893,B 20.7755,C -0.6437,E1 20.8091,E2 531.0392} C_DIS
LIN {X 16.9087,Y -126.066,Z 148,A -84.4183,B 20.7747,C -0.6686,E1 20.8062,E2 532.097} C_DIS
LIN {X 13.0707,Y -126.5221,Z 148,A -86.4095,B 20.7751,C -0.6572,E1 20.8006,E2 534.1185} C_DIS
LIN {X 7.0785,Y -126.9991,Z 148,A -88.9808,B 20.7749,C -0.6617,E1 20.7935,E2 536.6757} C_DIS
LIN {X 1.2384,Y -127.1896,Z 148,A -91.7512,B 20.7751,C -0.6552,E1 20.7857,E2 539.4634} C_DIS
LIN {X 1.2384,Y -127.1896,Z 148,A -91.7512,B 20.7751,C -0.6552,E1 20.7857,E2 539.4634} C_DIS
Enddeposition()
LIN {X 0.9002,Y -126.2385,Z 148,A -91.1745,B 19.5818,C -0.518,E1 19.5899,E2 539.1604} C_DIS
Startdeposition()
$VEL.CP = VEL_PRINT
LIN {X 3.8264,Y -126.1848,Z 148,A -89.5056,B 19.5815,C -0.5315,E1 19.5947,E2 537.4516} C_DIS
LIN {X 6.9366,Y -126.0531,Z 148,A -88.1072,B 19.5815,C -0.5314,E1 19.5986,E2 536.0541} C_DIS
LIN {X 10.4421,Y -125.8099,Z 148,A -86.4206,B 19.5814,C -0.5357,E1 19.6033,E2 534.3558} C_DIS
LIN {X 13.9061,Y -125.4747,Z 148,A -84.9266,B 19.5814,C -0.5331,E1 19.6075,E2 532.8708} C_DIS
LIN {X 16.9683,Y -125.098,Z 148,A -83.5303,B 19.5814,C -0.5338,E1 19.6113,E2 531.4741} C_DIS
LIN {X 20.0179,Y -124.6471,Z 148,A -82.1234,B 19.5814,C -0.535,E1 19.6152,E2 530.0653} C_DIS
LIN {X 23.1077,Y -124.1108,Z 148,A -80.693,B 19.5814,C -0.5363,E1 19.6191,E2 528.6329} C_DIS
LIN {X 26.1416,Y -123.5069,Z 148,A -79.2942,B 19.5814,C -0.5373,E1 19.623,E2 527.2336} C_DIS
LIN {X 29.9262,Y -122.6443,Z 148,A -77.3864,B 19.5811,C -0.5447,E1 19.6282,E2 525.3074} C_DIS
LIN {X 33.8769,Y -121.6118,Z 148,A -75.5954,B 19.5811,C -0.5441,E1 19.633,E2 523.522} C_DIS
LIN {X 38.1214,Y -120.3491,Z 148,A -73.5427,B 19.5811,C -0.548,E1 19.6385,E2 521.4624} C_DIS
LIN {X 41.828,Y -119.1122,Z 148,A -71.7561,B 19.581,C -0.5506,E1 19.6432,E2 519.6726} C_DIS
LIN {X 45.4322,Y -117.7839,Z 148,A -70.032,B 19.581,C -0.5521,E1 19.6477,E2 517.949} C_DIS
LIN {X 49.7257,Y -116.0368,Z 148,A -68.0925,B 19.581,C -0.5484,E1 19.6527,E2 516.0265} C_DIS
LIN {X 52.5487,Y -114.7863,Z 148,A -66.6226,B 19.581,C -0.5532,E1 19.6565,E2 514.5472} C_DIS
LIN {X 55.7663,Y -113.257,Z 148,A -65.0142,B 19.5809,C -0.5553,E1 19.6605,E2 512.9379} C_DIS
LIN {X 58.8628,Y -111.6791,Z 148,A -63.5942,B 19.5809,C -0.5515,E1 19.664,E2 511.5345} C_DIS
LIN {X 62.2213,Y -109.846,Z 148,A -61.6232,B 19.5806,C -0.5639,E1 19.6689,E2 509.5343} C_DIS
LIN {X 66.1921,Y -107.4995,Z 148,A -59.6895,B 19.5806,C -0.5611,E1 19.6735,E2 507.6167} C_DIS
LIN {X 69.4713,Y -105.4099,Z 148,A -57.7823,B 19.5804,C -0.5702,E1 19.678,E2 505.6907} C_DIS
LIN {X 73.2948,Y -102.7881,Z 148,A -55.8355,B 19.5805,C -0.5679,E1 19.6824,E2 503.7596} C_DIS
LIN {X 76.4457,Y -100.4672,Z 148,A -53.9313,B 19.5803,C -0.5767,E1 19.6867,E2 501.8382} C_DIS
LIN {X 80.0813,Y -97.5938,Z 148,A -51.9129,B 19.5803,C -0.5776,E1 19.6911,E2 499.8269} C_DIS
LIN {X 83.323,Y -94.8416,Z 148,A -49.9074,B 19.58,C -0.5849,E1 19.6953,E2 497.81} C_DIS
LIN {X 86.4906,Y -91.9615,Z 148,A -48.0628,B 19.58,C -0.5853,E1 19.6991,E2 495.9743} C_DIS
LIN {X 89.2616,Y -89.275,Z 148,A -46.2371,B 19.5798,C -0.5924,E1 19.7027,E2 494.1375} C_DIS
LIN {X 92.2041,Y -86.232,Z 148,A -44.3569,B 19.5798,C -0.5953,E1 19.7063,E2 492.2593} C_DIS
LIN {X 95.0876,Y -83.0412,Z 148,A -42.482,B 19.5797,C -0.5969,E1 19.7098,E2 490.3906} C_DIS
LIN {X 97.5846,Y -80.0925,Z 148,A -40.6619,B 19.5795,C -0.6041,E1 19.7131,E2 488.5601} C_DIS
LIN {X 100.4748,Y -76.4357,Z 148,A -38.5504,B 19.5793,C -0.6094,E1 19.7167,E2 486.446} C_DIS
LIN {X 103.2158,Y -72.6911,Z 148,A -36.4648,B 19.5792,C -0.6141,E1 19.7201,E2 484.3597} C_DIS
LIN {X 105.818,Y -68.8481,Z 148,A -34.3753,B 19.579,C -0.6191,E1 19.7233,E2 482.269} C_DIS
LIN {X 108.28,Y -64.908,Z 148,A -32.2857,B 19.5789,C -0.6242,E1 19.7264,E2 480.1783} C_DIS
LIN {X 110.5484,Y -60.964,Z 148,A -30.362,B 19.5789,C -0.6241,E1 19.729,E2 478.268} C_DIS
LIN {X 112.0665,Y -58.125,Z 148,A -28.926,B 19.5788,C -0.6272,E1 19.7309,E2 476.8326} C_DIS
LIN {X 113.4556,Y -55.3635,Z 148,A -27.3729,B 19.5785,C -0.6375,E1 19.7328,E2 475.2599} C_DIS
LIN {X 115.105,Y -51.8456,Z 148,A -25.795,B 19.5785,C -0.6349,E1 19.7346,E2 473.7007} C_DIS
LIN {X 116.6316,Y -48.3139,Z 148,A -23.9052,B 19.5782,C -0.6461,E1 19.7367,E2 471.7916} C_DIS
LIN {X 118.0487,Y -44.7413,Z 148,A -22.1876,B 19.5781,C -0.6502,E1 19.7384,E2 470.0744} C_DIS
LIN {X 119.5173,Y -40.6595,Z 148,A -20.2677,B 19.5779,C -0.654,E1 19.7402,E2 468.1571} C_DIS
LIN {X 120.5786,Y -37.3909,Z 148,A -18.8272,B 19.5779,C -0.6538,E1 19.7414,E2 466.728} C_DIS
LIN {X 121.4583,Y -34.4259,Z 148,A -17.2713,B 19.5776,C -0.6644,E1 19.7426,E2 465.1523} C_DIS
LIN {X 122.6411,Y -29.9396,Z 148,A -15.3436,B 19.5776,C -0.6635,E1 19.7439,E2 463.242} C_DIS
LIN {X 123.3377,Y -26.9255,Z 148,A -13.9514,B 19.5775,C -0.6673,E1 19.7448,E2 461.8489} C_DIS
LIN {X 123.9603,Y -23.8952,Z 148,A -12.5513,B 19.5774,C -0.6715,E1 19.7455,E2 460.4471} C_DIS
LIN {X 124.5256,Y -20.7479,Z 148,A -11.1396,B 19.5773,C -0.6744,E1 19.7462,E2 459.0378} C_DIS
LIN {X 124.99,Y -17.7377,Z 148,A -9.7557,B 19.5771,C -0.6788,E1 19.7468,E2 457.6515} C_DIS
LIN {X 125.3824,Y -14.7116,Z 148,A -8.3816,B 19.577,C -0.6826,E1 19.7472,E2 456.2766} C_DIS
LIN {X 125.7317,Y -11.3649,Z 148,A -6.7095,B 19.5766,C -0.6934,E1 19.7477,E2 454.5854} C_DIS
LIN {X 126.0043,Y -7.749,Z 148,A -5.2152,B 19.5766,C -0.6923,E1 19.748,E2 453.1061} C_DIS
LIN {X 126.1841,Y -3.854,Z 148,A -3.3405,B 19.5763,C -0.7022,E1 19.7482,E2 451.2166} C_DIS
LIN {X 126.2449,Y 0.1758,Z 148,A -1.4853,B 19.5761,C -0.709,E1 19.7482,E2 449.3558} C_DIS
LIN {X 126.185,Y 3.8198,Z 148,A -0.0316,B 19.5762,C -0.7058,E1 19.7482,E2 447.9228} C_DIS
LIN {X 126.0462,Y 7.0688,Z 148,A 1.419,B 19.5761,C -0.7093,E1 19.7479,E2 446.473} C_DIS
LIN {X 125.8368,Y 10.1229,Z 148,A 2.9765,B 19.5757,C -0.7207,E1 19.7476,E2 444.8941} C_DIS
LIN {X 125.4756,Y 13.8982,Z 148,A 4.5186,B 19.5757,C -0.7185,E1 19.7471,E2 443.3702} C_DIS
LIN {X 125.0957,Y 16.9863,Z 148,A 6.0701,B 19.5754,C -0.7287,E1 19.7466,E2 441.8007} C_DIS
LIN {X 124.5164,Y 20.8028,Z 148,A 7.6647,B 19.5754,C -0.7275,E1 19.7459,E2 440.2217} C_DIS
LIN {X 123.9626,Y 23.883,Z 148,A 9.0718,B 19.5754,C -0.7313,E1 19.7451,E2 438.8143} C_DIS
LIN {X 123.3406,Y 26.9119,Z 148,A 10.5959,B 19.575,C -0.7405,E1 19.7443,E2 437.2744} C_DIS
LIN {X 122.4583,Y 30.6788,Z 148,A 12.3609,B 19.5748,C -0.7462,E1 19.7431,E2 435.5059} C_DIS
LIN {X 121.4561,Y 34.4336,Z 148,A 14.1206,B 19.5746,C -0.7513,E1 19.7418,E2 433.7444} C_DIS
LIN {X 120.159,Y 38.7164,Z 148,A 16.0093,B 19.5746,C -0.7513,E1 19.7402,E2 431.8696} C_DIS
LIN {X 118.8621,Y 42.5315,Z 148,A 17.7904,B 19.5744,C -0.7547,E1 19.7386,E2 430.0917} C_DIS
LIN {X 117.5653,Y 45.9946,Z 148,A 19.4774,B 19.5743,C -0.7598,E1 19.7369,E2 428.4017} C_DIS
LIN {X 116.0302,Y 49.7411,Z 148,A 21.4342,B 19.5739,C -0.7699,E1 19.7348,E2 426.4291} C_DIS
LIN {X 114.4445,Y 53.2877,Z 148,A 23.1653,B 19.5737,C -0.7735,E1 19.7328,E2 424.6997} C_DIS
LIN {X 112.7641,Y 56.7591,Z 148,A 24.8497,B 19.5737,C -0.7755,E1 19.7307,E2 423.021} C_DIS
LIN {X 110.9777,Y 60.1793,Z 148,A 26.6603,B 19.5734,C -0.7827,E1 19.7283,E2 421.2017} C_DIS
LIN {X 108.6763,Y 64.2424,Z 148,A 28.7686,B 19.5732,C -0.7878,E1 19.7253,E2 419.0926} C_DIS
LIN {X 106.251,Y 68.1781,Z 148,A 30.8545,B 19.573,C -0.7927,E1 19.7222,E2 417.0059} C_DIS
LIN {X 103.6751,Y 72.0346,Z 148,A 32.9438,B 19.5728,C -0.7973,E1 19.7189,E2 414.9164} C_DIS
LIN {X 101.2072,Y 75.4627,Z 148,A 34.7713,B 19.5728,C -0.7983,E1 19.7159,E2 413.0975} C_DIS
LIN {X 98.5591,Y 78.8905,Z 148,A 36.7285,B 19.5726,C -0.8026,E1 19.7126,E2 411.1396} C_DIS
LIN {X 96.0959,Y 81.8724,Z 148,A 38.4554,B 19.5726,C -0.8054,E1 19.7095,E2 409.4146} C_DIS
LIN {X 93.289,Y 85.0574,Z 148,A 40.3882,B 19.5723,C -0.81,E1 19.7059,E2 407.4796} C_DIS
LIN {X 90.6292,Y 87.8855,Z 148,A 42.1177,B 19.5723,C -0.8125,E1 19.7025,E2 405.7525} C_DIS
LIN {X 87.3273,Y 91.1672,Z 148,A 44.2316,B 19.572,C -0.8169,E1 19.6983,E2 403.6371} C_DIS
LIN {X 84.4974,Y 93.7967,Z 148,A 46.0586,B 19.5718,C -0.8234,E1 19.6945,E2 401.8005} C_DIS
LIN {X 81.2806,Y 96.597,Z 148,A 47.9068,B 19.5718,C -0.8236,E1 19.6906,E2 399.9611} C_DIS
LIN {X 78.2843,Y 99.0415,Z 148,A 49.7331,B 19.5715,C -0.8296,E1 19.6866,E2 398.1258} C_DIS
LIN {X 74.9054,Y 101.6204,Z 148,A 51.5817,B 19.5715,C -0.8298,E1 19.6825,E2 396.2854} C_DIS
LIN {X 71.4161,Y 104.1021,Z 148,A 53.5868,B 19.5713,C -0.8355,E1 19.6779,E2 394.2724} C_DIS
LIN {X 67.5413,Y 106.657,Z 148,A 55.6718,B 19.5712,C -0.838,E1 19.673,E2 392.189} C_DIS
LIN {X 63.5692,Y 109.0715,Z 148,A 57.785,B 19.5711,C -0.8412,E1 19.6679,E2 390.0748} C_DIS
LIN {X 59.4594,Y 111.3651,Z 148,A 59.7719,B 19.5711,C -0.8382,E1 19.6631,E2 388.1042} C_DIS
LIN {X 56.7548,Y 112.7663,Z 148,A 61.1378,B 19.5711,C -0.8394,E1 19.6597,E2 386.7398} C_DIS
LIN {X 53.2896,Y 114.4436,Z 148,A 62.8804,B 19.5711,C -0.8413,E1 19.6553,E2 384.9974} C_DIS
LIN {X 49.7405,Y 116.0304,Z 148,A 64.783,B 19.5707,C -0.8487,E1 19.6504,E2 383.0789} C_DIS
LIN {X 45.4372,Y 117.782,Z 148,A 66.736,B 19.5709,C -0.8448,E1 19.6454,E2 381.1434} C_DIS
LIN {X 41.8363,Y 119.1093,Z 148,A 68.4934,B 19.5709,C -0.847,E1 19.6408,E2 379.3842} C_DIS
LIN {X 38.1243,Y 120.3482,Z 148,A 70.2441,B 19.5708,C -0.8475,E1 19.6361,E2 377.6363} C_DIS
LIN {X 34.4357,Y 121.4555,Z 148,A 72.1567,B 19.5705,C -0.8552,E1 19.6309,E2 375.7051} C_DIS
LIN {X 29.9472,Y 122.6392,Z 148,A 74.2498,B 19.5705,C -0.856,E1 19.6253,E2 373.6139} C_DIS
LIN {X 26.143,Y 123.5066,Z 148,A 75.8542,B 19.5707,C -0.8505,E1 19.621,E2 372.0287} C_DIS
LIN {X 23.1091,Y 124.1106,Z 148,A 77.2533,B 19.5707,C -0.8509,E1 19.6171,E2 370.6304} C_DIS
LIN {X 20.061,Y 124.6402,Z 148,A 78.6734,B 19.5707,C -0.852,E1 19.6132,E2 369.2088} C_DIS
LIN {X 16.9916,Y 125.095,Z 148,A 80.0853,B 19.5706,C -0.8526,E1 19.6093,E2 367.7969} C_DIS
LIN {X 13.1214,Y 125.5591,Z 148,A 81.8263,B 19.5706,C -0.8519,E1 19.6045,E2 366.0596} C_DIS
LIN {X 10.0822,Y 125.8403,Z 148,A 83.2099,B 19.5706,C -0.852,E1 19.6006,E2 364.6767} C_DIS
LIN {X 6.9643,Y 126.0517,Z 148,A 84.6558,B 19.5706,C -0.8531,E1 19.5966,E2 363.2283} C_DIS
LIN {X 3.1174,Y 126.2045,Z 148,A 86.3744,B 19.5706,C -0.852,E1 19.5918,E2 361.5136} C_DIS
LIN {X -0.002,Y 126.2444,Z 148,A 87.8325,B 19.5706,C -0.8534,E1 19.5877,E2 360.0515} C_DIS
LIN {X -3.8449,Y 126.1843,Z 148,A 89.5432,B 19.5706,C -0.8518,E1 19.583,E2 358.3455} C_DIS
LIN {X -6.9287,Y 126.0535,Z 148,A 90.9424,B 19.5706,C -0.8513,E1 19.5791,E2 356.9472} C_DIS
LIN {X -10.0694,Y 125.8414,Z 148,A 92.562,B 19.5704,C -0.8579,E1 19.5745,E2 355.307} C_DIS
LIN {X -13.915,Y 125.4737,Z 148,A 94.1316,B 19.5707,C -0.8502,E1 19.5702,E2 353.7592} C_DIS
LIN {X -16.9836,Y 125.096,Z 148,A 95.5343,B 19.5707,C -0.8495,E1 19.5663,E2 352.3575} C_DIS
LIN {X -20.04,Y 124.6436,Z 148,A 96.9605,B 19.5707,C -0.8495,E1 19.5624,E2 350.9296} C_DIS
LIN {X -23.0874,Y 124.1147,Z 148,A 98.531,B 19.5705,C -0.8547,E1 19.558,E2 349.3413} C_DIS
LIN {X -26.92,Y 123.3389,Z 148,A 100.1334,B 19.5708,C -0.8469,E1 19.5537,E2 347.7598} C_DIS
LIN {X -30.6691,Y 122.4608,Z 148,A 102.0434,B 19.5706,C -0.8514,E1 19.5485,E2 345.8329} C_DIS
LIN {X -34.4204,Y 121.4598,Z 148,A 103.7904,B 19.5707,C -0.8492,E1 19.5438,E2 344.0891} C_DIS
LIN {X -38.1385,Y 120.3436,Z 148,A 105.422,B 19.571,C -0.8425,E1 19.5395,E2 342.4737} C_DIS
LIN {X -41.0759,Y 119.373,Z 148,A 106.8297,B 19.571,C -0.841,E1 19.5357,E2 341.0669} C_DIS
LIN {X -43.989,Y 118.3305,Z 148,A 108.2379,B 19.5711,C -0.8395,E1 19.532,E2 339.6597} C_DIS
LIN {X -47.6103,Y 116.9209,Z 148,A 110.1673,B 19.571,C -0.8433,E1 19.527,E2 337.7134} C_DIS
LIN {X -51.8395,Y 115.1077,Z 148,A 112.1125,B 19.5713,C -0.8352,E1 19.5221,E2 335.7864} C_DIS
LIN {X -55.36,Y 113.4574,Z 148,A 113.943,B 19.5713,C -0.835,E1 19.5174,E2 333.9505} C_DIS
LIN {X -58.1314,Y 112.0631,Z 148,A 115.4108,B 19.5713,C -0.835,E1 19.5138,E2 332.4776} C_DIS
LIN {X -62.1254,Y 109.9001,Z 148,A 117.4928,B 19.5714,C -0.8323,E1 19.5087,E2 330.3956} C_DIS
LIN {X -65.5414,Y 107.8976,Z 148,A 119.3342,B 19.5714,C -0.8308,E1 19.5043,E2 328.5514} C_DIS
LIN {X -68.8452,Y 105.8199,Z 148,A 121.1099,B 19.5716,C -0.8277,E1 19.5001,E2 326.7773} C_DIS
LIN {X -72.6989,Y 103.2103,Z 148,A 123.227,B 19.5718,C -0.8239,E1 19.4953,E2 324.6622} C_DIS
LIN {X -76.4265,Y 100.4818,Z 148,A 125.333,B 19.5719,C -0.8201,E1 19.4905,E2 322.558} C_DIS
LIN {X -79.78,Y 97.84,Z 148,A 127.2059,B 19.5722,C -0.8138,E1 19.4865,E2 320.6948} C_DIS
LIN {X -82.7531,Y 95.339,Z 148,A 129.0551,B 19.5722,C -0.8131,E1 19.4825,E2 318.8383} C_DIS
LIN {X -86.1558,Y 92.2751,Z 148,A 131.0396,B 19.5725,C -0.8051,E1 19.4785,E2 316.8671} C_DIS
LIN {X -88.9992,Y 89.5357,Z 148,A 132.8597,B 19.5726,C -0.802,E1 19.4749,E2 315.0463} C_DIS
LIN {X -91.6995,Y 86.7683,Z 148,A 134.6405,B 19.5728,C -0.7988,E1 19.4714,E2 313.2651} C_DIS
LIN {X -94.2928,Y 83.9435,Z 148,A 136.4753,B 19.5728,C -0.798,E1 19.468,E2 311.4221} C_DIS
LIN {X -97.0949,Y 80.6854,Z 148,A 138.3562,B 19.5731,C -0.7907,E1 19.4646,E2 309.5519} C_DIS
LIN {X -99.5287,Y 77.664,Z 148,A 140.2155,B 19.5731,C -0.7897,E1 19.4614,E2 307.6841} C_DIS
LIN {X -102.3108,Y 73.9596,Z 148,A 142.3273,B 19.5733,C -0.7845,E1 19.4579,E2 305.5744} C_DIS
LIN {X -104.6838,Y 70.561,Z 148,A 144.1701,B 19.5736,C -0.7782,E1 19.455,E2 303.7387} C_DIS
LIN {X -107.0783,Y 66.8714,Z 148,A 146.2263,B 19.5736,C -0.7749,E1 19.4519,E2 301.6787} C_DIS
LIN {X -109.457,Y 62.9032,Z 148,A 148.3519,B 19.5739,C -0.77,E1 19.4489,E2 299.5535} C_DIS
LIN {X -111.3362,Y 59.5132,Z 148,A 149.9833,B 19.5742,C -0.7605,E1 19.4467,E2 297.9391} C_DIS
LIN {X -112.7587,Y 56.7698,Z 148,A 151.3779,B 19.5744,C -0.7563,E1 19.445,E2 296.5474} C_DIS
LIN {X -114.4309,Y 53.3172,Z 148,A 153.1432,B 19.5745,C -0.7521,E1 19.4428,E2 294.7822} C_DIS
LIN {X -115.7315,Y 50.4319,Z 148,A 154.7291,B 19.5745,C -0.7531,E1 19.441,E2 293.1817} C_DIS
LIN {X -117.5071,Y 46.1443,Z 148,A 156.6826,B 19.5749,C -0.7416,E1 19.439,E2 291.2485} C_DIS
LIN {X -118.6119,Y 43.2256,Z 148,A 158.1101,B 19.5751,C -0.7378,E1 19.4376,E2 289.822} C_DIS
LIN {X -119.8704,Y 39.6007,Z 148,A 160.0202,B 19.5751,C -0.7384,E1 19.4359,E2 287.8957} C_DIS
LIN {X -121.0188,Y 35.941,Z 148,A 161.6356,B 19.5754,C -0.7287,E1 19.4346,E2 286.2972} C_DIS
LIN {X -122.0663,Y 32.2023,Z 148,A 163.5708,B 19.5754,C -0.7294,E1 19.4332,E2 284.3452} C_DIS
LIN {X -122.9987,Y 28.4344,Z 148,A 165.1921,B 19.5757,C -0.7191,E1 19.4321,E2 282.7424} C_DIS
LIN {X -123.6618,Y 25.395,Z 148,A 166.6155,B 19.5759,C -0.7151,E1 19.4313,E2 281.3199} C_DIS
LIN {X -124.2535,Y 22.3195,Z 148,A 168.0463,B 19.576,C -0.7111,E1 19.4306,E2 279.8902} C_DIS
LIN {X -124.7573,Y 19.3059,Z 148,A 169.4497,B 19.5761,C -0.7073,E1 19.43,E2 278.4871} C_DIS
LIN {X -125.2643,Y 15.6994,Z 148,A 171.1993,B 19.5762,C -0.7055,E1 19.4293,E2 276.7292} C_DIS
LIN {X -125.6349,Y 12.3728,Z 148,A 172.7818,B 19.5762,C -0.703,E1 19.4289,E2 275.1418} C_DIS
LIN {X -125.9586,Y 8.4883,Z 148,A 174.4433,B 19.5766,C -0.6937,E1 19.4285,E2 273.4952} C_DIS
LIN {X -126.1263,Y 5.438,Z 148,A 176.0103,B 19.5766,C -0.6957,E1 19.4283,E2 271.9098} C_DIS
LIN {X -126.2341,Y 1.5536,Z 148,A 177.6023,B 19.5769,C -0.6842,E1 19.4283,E2 270.3399} C_DIS
LIN {X -126.2212,Y -2.3301,Z 148,A 179.3696,B 19.5771,C -0.6789,E1 19.4283,E2 268.5746} C_DIS
LIN {X -126.1261,Y -5.4434,Z 148,A -179.2136,B 19.5773,C -0.6746,E1 19.4284,E2 267.1594} C_DIS
LIN {X -125.9582,Y -8.494,Z 148,A -177.7621,B 19.5773,C -0.6725,E1 19.4287,E2 265.7027} C_DIS
LIN {X -125.6354,Y -12.368,Z 148,A -175.8739,B 19.5773,C -0.6714,E1 19.4291,E2 263.803} C_DIS
LIN {X -125.1975,Y -16.2094,Z 148,A -174.2418,B 19.5777,C -0.6617,E1 19.4297,E2 262.1872} C_DIS
LIN {X -124.7568,Y -19.3093,Z 148,A -172.8198,B 19.5778,C -0.6574,E1 19.4303,E2 260.767} C_DIS
LIN {X -124.2526,Y -22.3245,Z 148,A -171.4089,B 19.5779,C -0.654,E1 19.4309,E2 259.3554} C_DIS
LIN {X -123.5536,Y -25.9256,Z 148,A -169.6495,B 19.5779,C -0.6522,E1 19.4319,E2 257.5877} C_DIS
LIN {X -122.6406,Y -29.9416,Z 148,A -167.6948,B 19.5781,C -0.6496,E1 19.4332,E2 255.6257} C_DIS
LIN {X -121.447,Y -34.4661,Z 148,A -165.546,B 19.5782,C -0.6442,E1 19.4348,E2 253.4768} C_DIS
LIN {X -120.3479,Y -38.1252,Z 148,A -163.9634,B 19.5786,C -0.6338,E1 19.4361,E2 251.9135} C_DIS
LIN {X -119.1275,Y -41.7839,Z 148,A -162.0357,B 19.5786,C -0.635,E1 19.4378,E2 249.968} C_DIS
LIN {X -117.7841,Y -45.4317,Z 148,A -160.2633,B 19.5786,C -0.6302,E1 19.4396,E2 248.1967} C_DIS
LIN {X -116.0309,Y -49.7393,Z 148,A -158.1338,B 19.5788,C -0.625,E1 19.4419,E2 246.0676} C_DIS
LIN {X -114.4453,Y -53.2861,Z 148,A -156.3766,B 19.579,C -0.6199,E1 19.4439,E2 244.3131} C_DIS
LIN {X -112.7621,Y -56.763,Z 148,A -154.7544,B 19.5793,C -0.6104,E1 19.4459,E2 242.7077} C_DIS
LIN {X -110.9764,Y -60.1816,Z 148,A -152.8297,B 19.5793,C -0.6119,E1 19.4484,E2 240.7651} C_DIS
LIN {X -108.6687,Y -64.2554,Z 148,A -150.8411,B 19.5795,C -0.6015,E1 19.4512,E2 238.7943} C_DIS
LIN {X -106.6585,Y -67.5389,Z 148,A -148.93,B 19.5795,C -0.6029,E1 19.454,E2 236.8662} C_DIS
LIN {X -104.1035,Y -71.4141,Z 148,A -146.873,B 19.5797,C -0.5959,E1 19.4572,E2 234.8169} C_DIS
LIN {X -101.8706,Y -74.5649,Z 148,A -145.0651,B 19.5797,C -0.5936,E1 19.4602,E2 233.0043} C_DIS
LIN {X -99.1393,Y -78.1598,Z 148,A -143.028,B 19.5799,C -0.5883,E1 19.4637,E2 230.9703} C_DIS
LIN {X -96.5979,Y -81.2796,Z 148,A -141.2293,B 19.5801,C -0.5831,E1 19.4669,E2 229.1763} C_DIS
LIN {X -93.7892,Y -84.5058,Z 148,A -139.1841,B 19.5801,C -0.5826,E1 19.4707,E2 227.1207} C_DIS
LIN {X -90.8553,Y -87.6519,Z 148,A -137.2499,B 19.5802,C -0.5777,E1 19.4744,E2 225.1901} C_DIS
LIN {X -87.6094,Y -90.8964,Z 148,A -135.2104,B 19.5804,C -0.5719,E1 19.4784,E2 223.157} C_DIS
LIN {X -84.5005,Y -93.7939,Z 148,A -133.1907,B 19.5804,C -0.5714,E1 19.4826,E2 221.128} C_DIS
LIN {X -81.2839,Y -96.5943,Z 148,A -131.3237,B 19.5806,C -0.5652,E1 19.4866,E2 219.27} C_DIS
LIN {X -78.2876,Y -99.0389,Z 148,A -129.4809,B 19.5806,C -0.5652,E1 19.4906,E2 217.4182} C_DIS
LIN {X -74.6959,Y -101.7744,Z 148,A -127.4469,B 19.5806,C -0.5612,E1 19.4951,E2 215.3868} C_DIS
LIN {X -71.4351,Y -104.089,Z 148,A -125.5959,B 19.5807,C -0.5595,E1 19.4994,E2 213.5325} C_DIS
LIN {X -67.5442,Y -106.6552,Z 148,A -123.4865,B 19.5808,C -0.556,E1 19.5043,E2 211.4247} C_DIS
LIN {X -63.5778,Y -109.0665,Z 148,A -121.3571,B 19.5808,C -0.5538,E1 19.5095,E2 209.2933} C_DIS
LIN {X -59.5051,Y -111.3406,Z 148,A -119.3734,B 19.5811,C -0.5461,E1 19.5143,E2 207.3255} C_DIS
LIN {X -56.7584,Y -112.7645,Z 148,A -117.9819,B 19.5811,C -0.5438,E1 19.5177,E2 205.9358} C_DIS
LIN {X -53.2937,Y -114.4418,Z 148,A -116.2283,B 19.5812,C -0.542,E1 19.5222,E2 204.1817} C_DIS
LIN {X -49.7384,Y -116.0313,Z 148,A -114.3147,B 19.5812,C -0.5456,E1 19.5271,E2 202.2516} C_DIS
LIN {X -45.4434,Y -117.7796,Z 148,A -112.3319,B 19.5812,C -0.5389,E1 19.5322,E2 200.283} C_DIS
LIN {X -41.8141,Y -119.117,Z 148,A -110.5816,B 19.5813,C -0.5372,E1 19.5368,E2 198.5334} C_DIS
LIN {X -38.1264,Y -120.3475,Z 148,A -108.8257,B 19.5813,C -0.5355,E1 19.5415,E2 196.7784} C_DIS
LIN {X -34.4393,Y -121.4545,Z 148,A -106.9055,B 19.5813,C -0.5408,E1 19.5467,E2 194.8382} C_DIS
LIN {X -29.9358,Y -122.642,Z 148,A -104.8033,B 19.5813,C -0.5391,E1 19.5523,E2 192.737} C_DIS
LIN {X -26.1467,Y -123.5058,Z 148,A -103.1977,B 19.5815,C -0.5322,E1 19.5567,E2 191.1495} C_DIS
LIN {X -23.1134,Y -124.1097,Z 148,A -101.7957,B 19.5815,C -0.5316,E1 19.5605,E2 189.7473} C_DIS
LIN {X -20.0568,Y -124.6409,Z 148,A -100.3678,B 19.5815,C -0.5319,E1 19.5645,E2 188.3169} C_DIS
LIN {X -16.9979,Y -125.0941,Z 148,A -98.9554,B 19.5815,C -0.5319,E1 19.5684,E2 186.9029} C_DIS
LIN {X -13.9163,Y -125.4736,Z 148,A -97.4116,B 19.5814,C -0.5368,E1 19.5727,E2 185.3432} C_DIS
LIN {X -10.0955,Y -125.8392,Z 148,A -95.8355,B 19.5815,C -0.5303,E1 19.577,E2 183.7856} C_DIS
LIN {X -6.9838,Y -126.0507,Z 148,A -94.3903,B 19.5815,C -0.5314,E1 19.5811,E2 182.3364} C_DIS
LIN {X -3.0953,Y -126.2052,Z 148,A -92.6564,B 19.5815,C -0.5303,E1 19.5859,E2 180.6054} C_DIS
LIN {X -0.0084,Y -126.2444,Z 148,A -91.2165,B 19.5815,C -0.532,E1 19.5899,E2 179.1604} C_DIS
LIN {X -0.0084,Y -126.2444,Z 148,A -91.2165,B 19.5815,C -0.532,E1 19.5899,E2 179.1604} C_DIS
Enddeposition()
LIN {X 0.9406,Y -132.2856,Z 149,A -92.378,B 24.9667,C -1.3331,E1 25.0025,E2 178.8597} C_DIS
Startdeposition()
$VEL.CP = VEL_PRINT
LIN {X -3.2566,Y -132.25,Z 149,A -94.9029,B 24.9685,C -1.2958,E1 24.9952,E2 181.473} C_DIS
LIN {X -7.0684,Y -132.1011,Z 149,A -96.625,B 24.9687,C -1.2921,E1 24.9904,E2 183.2043} C_DIS
LIN {X -11.1385,Y -131.8196,Z 149,A -98.285,B 24.9685,C -1.2977,E1 24.9858,E2 184.8519} C_DIS
LIN {X -14.6139,Y -131.4805,Z 149,A -99.9113,B 24.9687,C -1.292,E1 24.9812,E2 186.4926} C_DIS
LIN {X -18.6495,Y -130.9681,Z 149,A -101.5565,B 24.9684,C -1.2983,E1 24.9767,E2 188.1239} C_DIS
LIN {X -22.1054,Y -130.4297,Z 149,A -103.1681,B 24.9686,C -1.2938,E1 24.9722,E2 189.7477} C_DIS
LIN {X -26.2622,Y -129.6562,Z 149,A -104.9142,B 24.9684,C -1.2989,E1 24.9675,E2 191.4836} C_DIS
LIN {X -29.5841,Y -128.9388,Z 149,A -106.3766,B 24.9684,C -1.3001,E1 24.9635,E2 192.945} C_DIS
LIN {X -33.3769,Y -128.0114,Z 149,A -108.178,B 24.9686,C -1.2955,E1 24.9586,E2 194.7601} C_DIS
LIN {X -37.1114,Y -126.977,Z 149,A -109.7482,B 24.9682,C -1.3021,E1 24.9544,E2 196.3169} C_DIS
LIN {X -40.3039,Y -126,Z 149,A -111.1784,B 24.9682,C -1.3041,E1 24.9506,E2 197.7451} C_DIS
LIN {X -43.415,Y -124.9621,Z 149,A -112.5815,B 24.968,C -1.3061,E1 24.9469,E2 199.1459} C_DIS
LIN {X -46.3769,Y -123.8934,Z 149,A -113.9779,B 24.968,C -1.3057,E1 24.9432,E2 200.5461} C_DIS
LIN {X -49.4553,Y -122.697,Z 149,A -115.4314,B 24.968,C -1.306,E1 24.9394,E2 202.0022} C_DIS
LIN {X -52.6258,Y -121.3709,Z 149,A -116.897,B 24.968,C -1.3088,E1 24.9357,E2 203.4646} C_DIS
LIN {X -55.7135,Y -119.985,Z 149,A -118.3888,B 24.9679,C -1.3092,E1 24.9319,E2 204.9591} C_DIS
LIN {X -59.0391,Y -118.3852,Z 149,A -120.0716,B 24.968,C -1.3069,E1 24.9276,E2 206.6517} C_DIS
LIN {X -65.707,Y -114.8194,Z 149,A -122.9332,B 24.9668,C -1.3321,E1 24.9207,E2 209.4616} C_DIS
LIN {X -69.8991,Y -112.3164,Z 149,A -125.4657,B 24.9676,C -1.3143,E1 24.9146,E2 212.044} C_DIS
LIN {X -73.69,Y -109.8669,Z 149,A -127.4521,B 24.9676,C -1.316,E1 24.9099,E2 214.0331} C_DIS
LIN {X -77.3646,Y -107.3112,Z 149,A -129.409,B 24.9674,C -1.3184,E1 24.9054,E2 215.991} C_DIS
LIN {X -80.9164,Y -104.6586,Z 149,A -131.3203,B 24.9673,C -1.3223,E1 24.9012,E2 217.8998} C_DIS
LIN {X -84.4277,Y -101.847,Z 149,A -133.2668,B 24.9671,C -1.3261,E1 24.897,E2 219.8446} C_DIS
LIN {X -87.7832,Y -98.9698,Z 149,A -135.1688,B 24.9668,C -1.3305,E1 24.893,E2 221.7435} C_DIS
LIN {X -91.0133,Y -96.0081,Z 149,A -137.0799,B 24.9667,C -1.3339,E1 24.8891,E2 223.6545} C_DIS
LIN {X -94.1093,Y -92.9755,Z 149,A -138.9757,B 24.9665,C -1.337,E1 24.8853,E2 225.5508} C_DIS
LIN {X -96.9863,Y -89.9698,Z 149,A -140.7971,B 24.9664,C -1.3401,E1 24.8818,E2 227.3728} C_DIS
LIN {X -99.977,Y -86.635,Z 149,A -142.7603,B 24.9662,C -1.3435,E1 24.8782,E2 229.3367} C_DIS
LIN {X -102.7829,Y -83.2863,Z 149,A -144.6721,B 24.966,C -1.3471,E1 24.8748,E2 231.2489} C_DIS
LIN {X -105.5756,Y -79.7161,Z 149,A -146.611,B 24.9657,C -1.3531,E1 24.8715,E2 233.1826} C_DIS
LIN {X -108.0957,Y -76.2639,Z 149,A -148.4732,B 24.9655,C -1.3573,E1 24.8685,E2 235.0438} C_DIS
LIN {X -110.6519,Y -72.5058,Z 149,A -150.4742,B 24.9653,C -1.3609,E1 24.8654,E2 237.0463} C_DIS
LIN {X -113.0327,Y -68.7356,Z 149,A -152.3938,B 24.965,C -1.3667,E1 24.8626,E2 238.962} C_DIS
LIN {X -115.1862,Y -65.0622,Z 149,A -154.2726,B 24.9648,C -1.3701,E1 24.8599,E2 240.8426} C_DIS
LIN {X -117.1919,Y -61.3713,Z 149,A -155.9904,B 24.9643,C -1.3801,E1 24.8577,E2 242.5456} C_DIS
LIN {X -118.6918,Y -58.4176,Z 149,A -157.4433,B 24.9642,C -1.3833,E1 24.8559,E2 243.9985} C_DIS
LIN {X -120.1255,Y -55.4097,Z 149,A -158.8928,B 24.964,C -1.3872,E1 24.8542,E2 245.4467} C_DIS
LIN {X -121.5131,Y -52.2971,Z 149,A -160.4117,B 24.9638,C -1.3895,E1 24.8525,E2 246.9686} C_DIS
LIN {X -123.2526,Y -48.054,Z 149,A -162.448,B 24.9637,C -1.393,E1 24.8503,E2 249.0079} C_DIS
LIN {X -124.4715,Y -44.802,Z 149,A -163.8757,B 24.9632,C -1.4012,E1 24.849,E2 250.4241} C_DIS
LIN {X -125.5655,Y -41.6381,Z 149,A -165.3581,B 24.9631,C -1.4041,E1 24.8477,E2 251.9082} C_DIS
LIN {X -126.6572,Y -38.1922,Z 149,A -167.0249,B 24.9631,C -1.4041,E1 24.8463,E2 253.5846} C_DIS
LIN {X -127.7744,Y -34.2656,Z 149,A -168.7204,B 24.9626,C -1.4131,E1 24.845,E2 255.2685} C_DIS
LIN {X -128.6285,Y -30.9053,Z 149,A -170.2341,B 24.9624,C -1.4172,E1 24.844,E2 256.7811} C_DIS
LIN {X -129.5271,Y -26.897,Z 149,A -172.0866,B 24.9623,C -1.4193,E1 24.8429,E2 258.6394} C_DIS
LIN {X -130.2315,Y -23.2421,Z 149,A -173.6196,B 24.9618,C -1.4283,E1 24.8421,E2 260.1602} C_DIS
LIN {X -130.7856,Y -19.8922,Z 149,A -175.1588,B 24.9618,C -1.4298,E1 24.8415,E2 261.705} C_DIS
LIN {X -131.3746,Y -15.5302,Z 149,A -177.0652,B 24.9614,C -1.436,E1 24.8408,E2 263.608} C_DIS
LIN {X -131.9655,Y -9.2586,Z 149,A -179.8929,B 24.9611,C -1.4401,E1 24.8401,E2 266.4428} C_DIS
LIN {X -132.1917,Y -5.0854,Z 149,A 178.4081,B 24.9605,C -1.4514,E1 24.8399,E2 268.1252} C_DIS
LIN {X -132.2837,Y -1.424,Z 149,A 176.7648,B 24.9605,C -1.4538,E1 24.8398,E2 269.7726} C_DIS
LIN {X -132.2697,Y 2.2863,Z 149,A 175.1843,B 24.96,C -1.4604,E1 24.8398,E2 271.3468} C_DIS
LIN {X -132.1837,Y 5.2883,Z 149,A 173.9065,B 24.9597,C -1.4658,E1 24.84,E2 272.6195} C_DIS
LIN {X -131.9993,Y 8.7798,Z 149,A 172.1078,B 24.9602,C -1.4573,E1 24.8403,E2 274.4492} C_DIS
LIN {X -131.6661,Y 12.8275,Z 149,A 170.5361,B 24.9594,C -1.472,E1 24.8407,E2 275.9954} C_DIS
LIN {X -131.0146,Y 18.3245,Z 149,A 168.3409,B 24.9584,C -1.4895,E1 24.8414,E2 278.162} C_DIS
LIN {X -130.235,Y 23.2226,Z 149,A 165.9753,B 24.9586,C -1.4863,E1 24.8425,E2 280.5494} C_DIS
LIN {X -128.802,Y 30.1831,Z 149,A 162.9371,B 24.958,C -1.4982,E1 24.8442,E2 283.5772} C_DIS
LIN {X -127.7749,Y 34.264,Z 149,A 161.0679,B 24.9577,C -1.5019,E1 24.8455,E2 285.4483} C_DIS
LIN {X -126.7424,Y 37.9125,Z 149,A 159.2713,B 24.9579,C -1.4998,E1 24.847,E2 287.2603} C_DIS
LIN {X -125.5466,Y 41.6946,Z 149,A 157.6935,B 24.9572,C -1.512,E1 24.8483,E2 288.818} C_DIS
LIN {X -124.4589,Y 44.837,Z 149,A 156.2354,B 24.957,C -1.5157,E1 24.8496,E2 290.2756} C_DIS
LIN {X -123.2853,Y 47.9699,Z 149,A 154.7662,B 24.9568,C -1.5194,E1 24.8511,E2 291.7444} C_DIS
LIN {X -122.0542,Y 51.021,Z 149,A 153.3245,B 24.9565,C -1.523,E1 24.8526,E2 293.1854} C_DIS
LIN {X -120.6681,Y 54.2183,Z 149,A 151.8305,B 24.9562,C -1.5284,E1 24.8543,E2 294.6748} C_DIS
LIN {X -119.2525,Y 57.2649,Z 149,A 150.3589,B 24.956,C -1.5321,E1 24.8561,E2 296.1456} C_DIS
LIN {X -117.6637,Y 60.4636,Z 149,A 148.6837,B 24.9561,C -1.5307,E1 24.8582,E2 297.8332} C_DIS
LIN {X -115.4929,Y 64.5164,Z 149,A 146.6735,B 24.9558,C -1.5357,E1 24.8609,E2 299.842} C_DIS
LIN {X -113.2302,Y 68.4091,Z 149,A 144.7721,B 24.9553,C -1.5438,E1 24.8636,E2 301.7341} C_DIS
LIN {X -110.9981,Y 71.9743,Z 149,A 142.8362,B 24.9553,C -1.5436,E1 24.8665,E2 303.6802} C_DIS
LIN {X -109.0703,Y 74.8635,Z 149,A 141.4019,B 24.9549,C -1.5512,E1 24.8687,E2 305.1035} C_DIS
LIN {X -106.4257,Y 78.5781,Z 149,A 139.3967,B 24.9547,C -1.5553,E1 24.872,E2 307.1088} C_DIS
LIN {X -103.7408,Y 82.0904,Z 149,A 137.3261,B 24.9548,C -1.553,E1 24.8756,E2 309.1945} C_DIS
LIN {X -100.9265,Y 85.5263,Z 149,A 134.9833,B 24.9557,C -1.5382,E1 24.8799,E2 311.5834} C_DIS
LIN {X -97.5752,Y 89.3309,Z 149,A 133.444,B 24.9535,C -1.5752,E1 24.8826,E2 313.0414} C_DIS
LIN {X -93.2891,Y 93.7977,Z 149,A 131.0195,B 24.9524,C -1.5943,E1 24.8873,E2 315.4309} C_DIS
LIN {X -89.7618,Y 97.1791,Z 149,A 128.5044,B 24.9532,C -1.5801,E1 24.8924,E2 317.9902} C_DIS
LIN {X -86.487,Y 100.1045,Z 149,A 126.5851,B 24.953,C -1.5837,E1 24.8965,E2 319.9085} C_DIS
LIN {X -83.0437,Y 102.9786,Z 149,A 124.6767,B 24.9526,C -1.5897,E1 24.9006,E2 321.8098} C_DIS
LIN {X -79.5962,Y 105.6661,Z 149,A 122.7627,B 24.9525,C -1.5928,E1 24.9048,E2 323.7234} C_DIS
LIN {X -76.2674,Y 108.0932,Z 149,A 120.9119,B 24.9525,C -1.5933,E1 24.909,E2 325.5794} C_DIS
LIN {X -73.3877,Y 110.0687,Z 149,A 119.4562,B 24.9521,C -1.5991,E1 24.9124,E2 327.0263} C_DIS
LIN {X -69.653,Y 112.4696,Z 149,A 117.4885,B 24.952,C -1.6006,E1 24.917,E2 328.9966} C_DIS
LIN {X -65.8582,Y 114.7331,Z 149,A 115.6589,B 24.9515,C -1.6082,E1 24.9214,E2 330.8135} C_DIS
LIN {X -62.9373,Y 116.361,Z 149,A 114.1363,B 24.9516,C -1.6071,E1 24.9251,E2 332.3431} C_DIS
LIN {X -59.9529,Y 117.9237,Z 149,A 112.7541,B 24.9512,C -1.6134,E1 24.9285,E2 333.7141} C_DIS
LIN {X -56.9016,Y 119.426,Z 149,A 111.2917,B 24.951,C -1.6163,E1 24.9322,E2 335.1734} C_DIS
LIN {X -53.7909,Y 120.8593,Z 149,A 109.8303,B 24.9508,C -1.6197,E1 24.9359,E2 336.6305} C_DIS
LIN {X -50.8651,Y 122.1193,Z 149,A 108.4228,B 24.9508,C -1.6203,E1 24.9395,E2 338.0396} C_DIS
LIN {X -47.7259,Y 123.3802,Z 149,A 106.9711,B 24.9506,C -1.623,E1 24.9433,E2 339.488} C_DIS
LIN {X -44.7174,Y 124.502,Z 149,A 105.5659,B 24.9506,C -1.6241,E1 24.947,E2 340.8935} C_DIS
LIN {X -41.4507,Y 125.6278,Z 149,A 104.0469,B 24.9506,C -1.6249,E1 24.951,E2 342.4136} C_DIS
LIN {X -37.6857,Y 126.8088,Z 149,A 102.2504,B 24.9506,C -1.6225,E1 24.9558,E2 344.2187} C_DIS
LIN {X -34.1226,Y 127.8126,Z 149,A 100.7098,B 24.9504,C -1.6273,E1 24.96,E2 345.7502} C_DIS
LIN {X -30.3517,Y 128.7619,Z 149,A 98.8632,B 24.9508,C -1.6209,E1 24.965,E2 347.6147} C_DIS
LIN {X -26.468,Y 129.6144,Z 149,A 97.3028,B 24.9502,C -1.6305,E1 24.9692,E2 349.1543} C_DIS
LIN {X -22.8675,Y 130.2985,Z 149,A 95.749,B 24.95,C -1.6334,E1 24.9735,E2 350.7028} C_DIS
LIN {X -15.7147,Y 131.3526,Z 149,A 92.583,B 24.95,C -1.6337,E1 24.9822,E2 353.8706} C_DIS
LIN {X -11.9025,Y 131.7549,Z 149,A 90.7956,B 24.9503,C -1.6281,E1 24.9872,E2 355.6723} C_DIS
LIN {X -8.0287,Y 132.0456,Z 149,A 89.2075,B 24.95,C -1.6336,E1 24.9916,E2 357.2479} C_DIS
LIN {X -3.7845,Y 132.2353,Z 149,A 87.3555,B 24.95,C -1.6336,E1 24.9968,E2 359.1003} C_DIS
LIN {X 0.4789,Y 132.2889,Z 149,A 85.5268,B 24.95,C -1.6349,E1 25.0019,E2 360.9259} C_DIS
LIN {X 4.2317,Y 132.2229,Z 149,A 83.8108,B 24.9502,C -1.6305,E1 25.0067,E2 362.6521} C_DIS
LIN {X 8.1573,Y 132.0377,Z 149,A 82.2117,B 24.9499,C -1.6357,E1 25.0111,E2 364.238} C_DIS
LIN {X 12.0905,Y 131.7368,Z 149,A 80.4255,B 24.9501,C -1.6316,E1 25.0161,E2 366.033} C_DIS
LIN {X 15.8457,Y 131.337,Z 149,A 78.895,B 24.9498,C -1.6367,E1 25.0203,E2 367.5504} C_DIS
LIN {X 19.3262,Y 130.8714,Z 149,A 77.2415,B 24.9502,C -1.6295,E1 25.025,E2 369.2194} C_DIS
LIN {X 23.2943,Y 130.2222,Z 149,A 75.6254,B 24.9499,C -1.6353,E1 25.0294,E2 370.8201} C_DIS
LIN {X 26.4948,Y 129.6089,Z 149,A 74.2159,B 24.9499,C -1.6348,E1 25.0332,E2 372.2292} C_DIS
LIN {X 29.6689,Y 128.9194,Z 149,A 72.76,B 24.9501,C -1.6315,E1 25.0372,E2 373.6909} C_DIS
LIN {X 35.4045,Y 127.4636,Z 149,A 70.4817,B 24.9493,C -1.6446,E1 25.0433,E2 375.9348} C_DIS
LIN {X 39.8015,Y 126.1604,Z 149,A 68.2014,B 24.9503,C -1.6278,E1 25.0495,E2 378.2507} C_DIS
LIN {X 43.3021,Y 125.0012,Z 149,A 66.6643,B 24.9503,C -1.6295,E1 25.0535,E2 379.7808} C_DIS
LIN {X 46.4751,Y 123.8566,Z 149,A 65.2083,B 24.9503,C -1.6284,E1 25.0573,E2 381.2364} C_DIS
LIN {X 49.5598,Y 122.6548,Z 149,A 63.7872,B 24.9503,C -1.6276,E1 25.061,E2 382.6562} C_DIS
LIN {X 52.604,Y 121.3804,Z 149,A 62.3204,B 24.9506,C -1.6241,E1 25.0648,E2 384.128} C_DIS
LIN {X 56.0985,Y 119.807,Z 149,A 60.6289,B 24.9508,C -1.6204,E1 25.0691,E2 385.8238} C_DIS
LIN {X 59.7413,Y 118.0314,Z 149,A 58.6005,B 24.9518,C -1.6039,E1 25.0742,E2 387.8857} C_DIS
LIN {X 62.9767,Y 116.3398,Z 149,A 57.3825,B 24.9508,C -1.6206,E1 25.0771,E2 389.0607} C_DIS
LIN {X 66.2451,Y 114.5096,Z 149,A 55.6698,B 24.9512,C -1.6135,E1 25.0813,E2 390.785} C_DIS
LIN {X 70.1469,Y 112.1622,Z 149,A 53.6795,B 24.9515,C -1.6095,E1 25.0861,E2 392.7786} C_DIS
LIN {X 73.8601,Y 109.7528,Z 149,A 51.7781,B 24.9516,C -1.6072,E1 25.0905,E2 394.6792} C_DIS
LIN {X 77.3897,Y 107.293,Z 149,A 49.9057,B 24.9518,C -1.6034,E1 25.0948,E2 396.554} C_DIS
LIN {X 80.9822,Y 104.6076,Z 149,A 48.0004,B 24.9519,C -1.6018,E1 25.099,E2 398.4561} C_DIS
LIN {X 84.4277,Y 101.847,Z 149,A 46.0944,B 24.9521,C -1.5985,E1 25.1031,E2 400.3628} C_DIS
LIN {X 87.6322,Y 99.1032,Z 149,A 44.1656,B 24.9527,C -1.5894,E1 25.1072,E2 402.3055} C_DIS
LIN {X 92.0249,Y 95.0383,Z 149,A 41.7381,B 24.9525,C -1.5927,E1 25.1121,E2 404.7153} C_DIS
LIN {X 94.9169,Y 92.1502,Z 149,A 39.9205,B 24.9529,C -1.5862,E1 25.1157,E2 406.5404} C_DIS
LIN {X 97.8928,Y 88.9825,Z 149,A 38.0406,B 24.9531,C -1.5821,E1 25.1193,E2 408.4218} C_DIS
LIN {X 100.0671,Y 86.5303,Z 149,A 35.4584,B 24.9569,C -1.5171,E1 25.1243,E2 411.1455} C_DIS
LIN {X 105.3104,Y 80.0669,Z 149,A 33.3482,B 24.9528,C -1.5876,E1 25.1276,E2 413.0795} C_DIS
LIN {X 108.2195,Y 76.0883,Z 149,A 30.9359,B 24.954,C -1.5672,E1 25.1315,E2 415.5283} C_DIS
LIN {X 110.7176,Y 72.406,Z 149,A 29.0182,B 24.9543,C -1.5626,E1 25.1345,E2 417.4473} C_DIS
LIN {X 113.0014,Y 68.7874,Z 149,A 27.1585,B 24.9546,C -1.5572,E1 25.1373,E2 419.3102} C_DIS
LIN {X 115.2066,Y 65.0259,Z 149,A 25.273,B 24.9549,C -1.5522,E1 25.1399,E2 421.1979} C_DIS
LIN {X 117.2452,Y 61.2697,Z 149,A 23.5411,B 24.9548,C -1.5534,E1 25.1421,E2 422.9177} C_DIS
LIN {X 118.8217,Y 58.1544,Z 149,A 22.0613,B 24.9549,C -1.5509,E1 25.144,E2 424.3957} C_DIS
LIN {X 120.1509,Y 55.3548,Z 149,A 20.7068,B 24.9552,C -1.5463,E1 25.1456,E2 425.7536} C_DIS
LIN {X 121.619,Y 52.052,Z 149,A 19.0218,B 24.9558,C -1.5352,E1 25.1475,E2 427.4555} C_DIS
LIN {X 123.2284,Y 48.1162,Z 149,A 17.2962,B 24.9558,C -1.536,E1 25.1493,E2 429.1697} C_DIS
LIN {X 124.4773,Y 44.786,Z 149,A 15.7876,B 24.956,C -1.5331,E1 25.1507,E2 430.6768} C_DIS
LIN {X 125.5485,Y 41.689,Z 149,A 14.392,B 24.9561,C -1.53,E1 25.152,E2 432.0717} C_DIS
LIN {X 126.5001,Y 38.7056,Z 149,A 13.0362,B 24.9564,C -1.5258,E1 25.1531,E2 433.4297} C_DIS
LIN {X 127.4376,Y 35.4977,Z 149,A 11.5981,B 24.9566,C -1.5218,E1 25.1542,E2 434.8689} C_DIS
LIN {X 128.2961,Y 32.2584,Z 149,A 10.1205,B 24.957,C -1.5158,E1 25.1552,E2 436.3522} C_DIS
LIN {X 129.2712,Y 28.0965,Z 149,A 8.2886,B 24.9572,C -1.511,E1 25.1564,E2 438.1849} C_DIS
LIN {X 130.0237,Y 24.3821,Z 149,A 6.5973,B 24.9577,C -1.503,E1 25.1573,E2 439.8851} C_DIS
LIN {X 130.7133,Y 20.3593,Z 149,A 4.9137,B 24.9577,C -1.5019,E1 25.158,E2 441.5613} C_DIS
LIN {X 131.267,Y 16.4322,Z 149,A 3.0851,B 24.9584,C -1.4902,E1 25.1587,E2 443.4068} C_DIS
LIN {X 131.6911,Y 12.5672,Z 149,A 1.5414,B 24.9583,C -1.4924,E1 25.1592,E2 444.9361} C_DIS
LIN {X 132.0129,Y 8.5587,Z 149,A -0.2352,B 24.9587,C -1.4848,E1 25.1595,E2 446.7202} C_DIS
LIN {X 132.2022,Y 4.8152,Z 149,A -1.8672,B 24.959,C -1.479,E1 25.1597,E2 448.3562} C_DIS
LIN {X 132.2905,Y 0.4939,Z 149,A -3.7027,B 24.9593,C -1.4748,E1 25.1597,E2 450.1906} C_DIS
LIN {X 132.2416,Y -3.5603,Z 149,A -5.4067,B 24.9594,C -1.4718,E1 25.1597,E2 451.8914} C_DIS
LIN {X 132.0854,Y -7.3806,Z 149,A -7.1689,B 24.96,C -1.4605,E1 25.1595,E2 453.6699} C_DIS
LIN {X 131.8106,Y -11.2448,Z 149,A -8.7046,B 24.96,C -1.4628,E1 25.1591,E2 455.1911} C_DIS
LIN {X 131.4306,Y -15.0609,Z 149,A -10.4588,B 24.9605,C -1.4521,E1 25.1586,E2 456.9601} C_DIS
LIN {X 130.9478,Y -18.7915,Z 149,A -11.9764,B 24.9605,C -1.4529,E1 25.158,E2 458.4669} C_DIS
LIN {X 130.3341,Y -22.6687,Z 149,A -13.7671,B 24.961,C -1.4423,E1 25.1572,E2 460.272} C_DIS
LIN {X 129.6233,Y -26.4239,Z 149,A -15.3129,B 24.961,C -1.4429,E1 25.1564,E2 461.8074} C_DIS
LIN {X 128.9277,Y -29.6325,Z 149,A -16.6564,B 24.961,C -1.4425,E1 25.1556,E2 463.1439} C_DIS
LIN {X 128.225,Y -32.5384,Z 149,A -18.0185,B 24.9614,C -1.4346,E1 25.1546,E2 464.5168} C_DIS
LIN {X 127.328,Y -35.8895,Z 149,A -19.4954,B 24.9616,C -1.4311,E1 25.1536,E2 465.9934} C_DIS
LIN {X 125.81,Y -40.8984,Z 149,A -21.7051,B 24.9619,C -1.4269,E1 25.1517,E2 468.2005} C_DIS
LIN {X 124.95,Y -43.45,Z 149,A -22.9087,B 24.9622,C -1.4212,E1 25.1506,E2 469.4109} C_DIS
LIN {X 123.8397,Y -46.5202,Z 149,A -24.3164,B 24.9624,C -1.417,E1 25.1493,E2 470.8204} C_DIS
LIN {X 122.6138,Y -49.6617,Z 149,A -25.7495,B 24.9626,C -1.4139,E1 25.1478,E2 472.2529} C_DIS
LIN {X 121.3622,Y -52.646,Z 149,A -27.1494,B 24.9628,C -1.4096,E1 25.1463,E2 473.6553} C_DIS
LIN {X 120.0163,Y -55.6459,Z 149,A -28.5586,B 24.963,C -1.406,E1 25.1446,E2 475.0653} C_DIS
LIN {X 118.4365,Y -58.9351,Z 149,A -30.2241,B 24.9635,C -1.3965,E1 25.1426,E2 476.7444} C_DIS
LIN {X 115.8197,Y -63.9272,Z 149,A -32.3089,B 24.9628,C -1.4086,E1 25.1399,E2 478.7896} C_DIS
LIN {X 113.4127,Y -68.1071,Z 149,A -34.7355,B 24.9641,C -1.3839,E1 25.1364,E2 481.262} C_DIS
LIN {X 111.167,Y -71.714,Z 149,A -36.5916,B 24.9644,C -1.3776,E1 25.1336,E2 483.1235} C_DIS
LIN {X 108.6984,Y -75.4027,Z 149,A -38.4687,B 24.9646,C -1.3746,E1 25.1307,E2 484.9985} C_DIS
Enddeposition()
END
